(* IEC 61131-3 sources: TIA2AX/tests/test_projects/expected/HW_2200330_V18/ST40_PLC, 6 files *)

(* ---- HwInputs.st ---- *)
TYPE
	HwInputs : STRUCT
		ST40_2_DM260_Acquisition_Status_1 AT %B2500 : ARRAY[0..2] OF BYTE;
		ST40_2_DM260_Results_Status_1 AT %B2503 : BYTE;
		ST40_2_DM260_Soft_Event_Control_1 AT %B2504 : BYTE;
		ST40_2_DM260_Result_Data_64_bytes_1 AT %B2510 : ARRAY[0..71] OF BYTE;
		ST40_3_DM260_Acquisition_Status_1 AT %B3500 : ARRAY[0..2] OF BYTE;
		ST40_3_DM260_Results_Status_1 AT %B3503 : BYTE;
		ST40_3_DM260_Soft_Event_Control_1 AT %B3504 : BYTE;
		ST40_3_DM260_Result_Data_64_bytes_1 AT %B3510 : ARRAY[0..71] OF BYTE;
		ST40_1_DM260_Acquisition_Status_1 AT %B1600 : ARRAY[0..2] OF BYTE;
		ST40_1_DM260_Results_Status_1 AT %B1603 : BYTE;
		ST40_1_DM260_Soft_Event_Control_1 AT %B1604 : BYTE;
		ST40_1_DM260_Result_Data_64_bytes_1 AT %B1610 : ARRAY[0..71] OF BYTE;
		ST40_2_Promess_Menu_30_01_In_1 AT %B2100 : WORD;
		ST40_2_Promess_Menu_30_02_In_1 AT %B2102 : WORD;
		ST40_2_Promess_Menu_30_03_In_1 AT %B2104 : WORD;
		ST40_2_Promess_Menu_30_04_In_1 AT %B2106 : WORD;
		ST40_2_Promess_Menu_30_05_In_1 AT %B2108 : WORD;
		ST40_2_Promess_Menu_30_06_In_1 AT %B2110 : WORD;
		ST40_2_Promess_Menu_30_07_In_1 AT %B2112 : WORD;
		ST40_2_Promess_Menu_30_08_In_1 AT %B2114 : WORD;
		ST40_2_Promess_Menu_30_09_In_1 AT %B2116 : WORD;
		ST40_2_Promess_Menu_30_10_In_1 AT %B2118 : WORD;
		ST40_2_Promess_Menu_30_11_In_1 AT %B2120 : WORD;
		ST40_2_Promess_Menu_30_12_In_1 AT %B2122 : WORD;
		ST40_2_Promess_Menu_30_13_In_1 AT %B2124 : WORD;
		ST40_2_Promess_Menu_30_14_In_1 AT %B2126 : WORD;
		ST40_2_Promess_Menu_30_15_In_1 AT %B2128 : WORD;
		ST40_2_Promess_Menu_30_16_In_1 AT %B2130 : WORD;
		ST40_2_Promess_Menu_30_17_In_1 AT %B2132 : WORD;
		ST40_2_Promess_Menu_30_18_In_1 AT %B2134 : WORD;
		ST40_2_Promess_Menu_30_19_In_1 AT %B2136 : WORD;
		ST40_2_Promess_Menu_30_20_In_1 AT %B2138 : WORD;
		ST40_2_Promess_Menu_30_21_In_1 AT %B2140 : WORD;
		ST40_2_Promess_Menu_30_22_In_1 AT %B2142 : WORD;
		ST40_2_Promess_Menu_30_23_In_1 AT %B2144 : WORD;
		ST40_2_Promess_Menu_30_24_In_1 AT %B2146 : WORD;
		ST40_2_Promess_Menu_30_25_In_1 AT %B2148 : WORD;
		ST40_2_Promess_Menu_30_26_In_1 AT %B2150 : WORD;
		ST40_2_Promess_Menu_30_27_In_1 AT %B2152 : WORD;
		ST40_2_Promess_Menu_30_28_In_1 AT %B2154 : WORD;
		ST40_2_Promess_Menu_30_29_In_1 AT %B2156 : WORD;
		ST40_2_Promess_Menu_30_30_In_1 AT %B2158 : WORD;
		ST40_2_Promess_Menu_30_31_In_1 AT %B2160 : WORD;
		ST40_2_Promess_Menu_30_32_In_1 AT %B2162 : WORD;
		ST40_ET200SP_CM_4xIO_Link_1 AT %B100 : ARRAY[0..31] OF BYTE;
		ST40_ET200SP_CM_4xIO_Link_2 AT %B132 : ARRAY[0..31] OF BYTE;
		ST40_ET200SP_DI_8x24VDC_ST_1 AT %B0 : BYTE;
		ST40_ET200SP_DI_8x24VDC_ST_2 AT %B1 : BYTE;
		ST40_ET200SP_DI_16x24VDC_ST_1 AT %B2 : WORD;
		ST40_ET200SP_DI_8x24VDC_ST_3 AT %B4 : BYTE;
	END_STRUCT;
END_TYPE

(* ---- HwOutputs.st ---- *)
TYPE
	HwOutputs : STRUCT
		ST40_2_DM260_Acquisition_Control_1 AT %B2500 : BYTE;
		ST40_2_DM260_Results_Control_1 AT %B2503 : BYTE;
		ST40_2_DM260_Soft_Event_Control_1 AT %B2504 : BYTE;
		ST40_2_DM260_User_Data_64_bytes_1 AT %B2510 : ARRAY[0..67] OF BYTE;
		ST40_3_DM260_Acquisition_Control_1 AT %B3500 : BYTE;
		ST40_3_DM260_Results_Control_1 AT %B3503 : BYTE;
		ST40_3_DM260_Soft_Event_Control_1 AT %B3504 : BYTE;
		ST40_3_DM260_User_Data_64_bytes_1 AT %B3510 : ARRAY[0..67] OF BYTE;
		ST40_1_DM260_Acquisition_Control_1 AT %B1600 : BYTE;
		ST40_1_DM260_Results_Control_1 AT %B1603 : BYTE;
		ST40_1_DM260_Soft_Event_Control_1 AT %B1604 : BYTE;
		ST40_1_DM260_User_Data_64_bytes_1 AT %B1610 : ARRAY[0..67] OF BYTE;
		ST40_2_Promess_Menu_30_33_Out_1 AT %B2100 : WORD;
		ST40_2_Promess_Menu_30_34_Out_1 AT %B2102 : WORD;
		ST40_2_Promess_Menu_30_35_Out_1 AT %B2104 : WORD;
		ST40_2_Promess_Menu_30_36_Out_1 AT %B2106 : WORD;
		ST40_2_Promess_Menu_30_37_Out_1 AT %B2108 : WORD;
		ST40_2_Promess_Menu_30_38_Out_1 AT %B2110 : WORD;
		ST40_2_Promess_Menu_30_39_Out_1 AT %B2112 : WORD;
		ST40_2_Promess_Menu_30_40_Out_1 AT %B2114 : WORD;
		ST40_2_Promess_Menu_30_41_Out_1 AT %B2116 : WORD;
		ST40_2_Promess_Menu_30_42_Out_1 AT %B2118 : WORD;
		ST40_2_Promess_Menu_30_43_Out_1 AT %B2120 : WORD;
		ST40_2_Promess_Menu_30_44_Out_1 AT %B2122 : WORD;
		ST40_2_Promess_Menu_30_45_Out_1 AT %B2124 : WORD;
		ST40_2_Promess_Menu_30_46_Out_1 AT %B2126 : WORD;
		ST40_2_Promess_Menu_30_47_Out_1 AT %B2128 : WORD;
		ST40_2_Promess_Menu_30_48_Out_1 AT %B2130 : WORD;
		ST40_2_Promess_Menu_30_49_Out_1 AT %B2132 : WORD;
		ST40_2_Promess_Menu_30_50_Out_1 AT %B2134 : WORD;
		ST40_2_Promess_Menu_30_51_Out_1 AT %B2136 : WORD;
		ST40_2_Promess_Menu_30_52_Out_1 AT %B2138 : WORD;
		ST40_2_Promess_Menu_30_53_Out_1 AT %B2140 : WORD;
		ST40_2_Promess_Menu_30_54_Out_1 AT %B2142 : WORD;
		ST40_2_Promess_Menu_30_55_Out_1 AT %B2144 : WORD;
		ST40_2_Promess_Menu_30_56_Out_1 AT %B2146 : WORD;
		ST40_2_Promess_Menu_30_57_Out_1 AT %B2148 : WORD;
		ST40_2_Promess_Menu_30_58_Out_1 AT %B2150 : WORD;
		ST40_2_Promess_Menu_30_59_Out_1 AT %B2152 : WORD;
		ST40_2_Promess_Menu_30_60_Out_1 AT %B2154 : WORD;
		ST40_2_Promess_Menu_30_61_Out_1 AT %B2156 : WORD;
		ST40_2_Promess_Menu_30_62_Out_1 AT %B2158 : WORD;
		ST40_2_Promess_Menu_30_63_Out_1 AT %B2160 : WORD;
		ST40_2_Promess_Menu_30_64_Out_1 AT %B2162 : WORD;
		ST40_CPX_MPA1S_VMPA1_FB_EMS_8_8DO_1 AT %B200 : BYTE;
		ST40_CPX_MPA1S_VMPA1_FB_EMS_8_8DO_2 AT %B201 : BYTE;
		ST40_CPX_MPA1S_VMPA1_FB_EMS_8_8DO_3 AT %B202 : BYTE;
		ST40_CPX_MPA1G_VMPA1_FB_EMG_8_8DO_1 AT %B203 : BYTE;
		ST40_ET200SP_CM_4xIO_Link_1 AT %B100 : ARRAY[0..31] OF BYTE;
		ST40_ET200SP_CM_4xIO_Link_2 AT %B132 : ARRAY[0..31] OF BYTE;
		ST40_ET200SP_DQ_16x24VDC_0_5A_ST_1 AT %B0 : WORD;
		ST40_ET200SP_DQ_8x24VDC_0_5A_ST_2 AT %B2 : BYTE;
		ST40_ET200SP_DQ_8x24VDC_0_5A_ST_3 AT %B3 : BYTE;
	END_STRUCT;
END_TYPE

(* ---- PlcInputs.st ---- *)
TYPE
	PlcInputs : STRUCT
		ST40_2_DM260_Acquisition_Status_1 : ARRAY[0..2] OF BYTE;
		ST40_2_DM260_Results_Status_1 : BYTE;
		ST40_2_DM260_Soft_Event_Control_1 : BYTE;
		ST40_2_DM260_Result_Data_64_bytes_1 : ARRAY[0..71] OF BYTE;
		ST40_3_DM260_Acquisition_Status_1 : ARRAY[0..2] OF BYTE;
		ST40_3_DM260_Results_Status_1 : BYTE;
		ST40_3_DM260_Soft_Event_Control_1 : BYTE;
		ST40_3_DM260_Result_Data_64_bytes_1 : ARRAY[0..71] OF BYTE;
		ST40_1_DM260_Acquisition_Status_1 : ARRAY[0..2] OF BYTE;
		ST40_1_DM260_Results_Status_1 : BYTE;
		ST40_1_DM260_Soft_Event_Control_1 : BYTE;
		ST40_1_DM260_Result_Data_64_bytes_1 : ARRAY[0..71] OF BYTE;
		ST40_2_Promess_Menu_30_01_In_1 : WORD;
		ST40_2_Promess_Menu_30_02_In_1 : WORD;
		ST40_2_Promess_Menu_30_03_In_1 : WORD;
		ST40_2_Promess_Menu_30_04_In_1 : WORD;
		ST40_2_Promess_Menu_30_05_In_1 : WORD;
		ST40_2_Promess_Menu_30_06_In_1 : WORD;
		ST40_2_Promess_Menu_30_07_In_1 : WORD;
		ST40_2_Promess_Menu_30_08_In_1 : WORD;
		ST40_2_Promess_Menu_30_09_In_1 : WORD;
		ST40_2_Promess_Menu_30_10_In_1 : WORD;
		ST40_2_Promess_Menu_30_11_In_1 : WORD;
		ST40_2_Promess_Menu_30_12_In_1 : WORD;
		ST40_2_Promess_Menu_30_13_In_1 : WORD;
		ST40_2_Promess_Menu_30_14_In_1 : WORD;
		ST40_2_Promess_Menu_30_15_In_1 : WORD;
		ST40_2_Promess_Menu_30_16_In_1 : WORD;
		ST40_2_Promess_Menu_30_17_In_1 : WORD;
		ST40_2_Promess_Menu_30_18_In_1 : WORD;
		ST40_2_Promess_Menu_30_19_In_1 : WORD;
		ST40_2_Promess_Menu_30_20_In_1 : WORD;
		ST40_2_Promess_Menu_30_21_In_1 : WORD;
		ST40_2_Promess_Menu_30_22_In_1 : WORD;
		ST40_2_Promess_Menu_30_23_In_1 : WORD;
		ST40_2_Promess_Menu_30_24_In_1 : WORD;
		ST40_2_Promess_Menu_30_25_In_1 : WORD;
		ST40_2_Promess_Menu_30_26_In_1 : WORD;
		ST40_2_Promess_Menu_30_27_In_1 : WORD;
		ST40_2_Promess_Menu_30_28_In_1 : WORD;
		ST40_2_Promess_Menu_30_29_In_1 : WORD;
		ST40_2_Promess_Menu_30_30_In_1 : WORD;
		ST40_2_Promess_Menu_30_31_In_1 : WORD;
		ST40_2_Promess_Menu_30_32_In_1 : WORD;
		ST40_ET200SP_CM_4xIO_Link_1 : ARRAY[0..31] OF BYTE;
		ST40_ET200SP_CM_4xIO_Link_2 : ARRAY[0..31] OF BYTE;
		ST40_ET200SP_DI_8x24VDC_ST_1 : BYTE;
		ST40_ET200SP_DI_8x24VDC_ST_2 : BYTE;
		ST40_ET200SP_DI_16x24VDC_ST_1 : WORD;
		ST40_ET200SP_DI_8x24VDC_ST_3 : BYTE;
	END_STRUCT;
END_TYPE

(* ---- PlcOutputs.st ---- *)
TYPE
	PlcOutputs : STRUCT
		ST40_2_DM260_Acquisition_Control_1 : BYTE;
		ST40_2_DM260_Results_Control_1 : BYTE;
		ST40_2_DM260_Soft_Event_Control_1 : BYTE;
		ST40_2_DM260_User_Data_64_bytes_1 : ARRAY[0..67] OF BYTE;
		ST40_3_DM260_Acquisition_Control_1 : BYTE;
		ST40_3_DM260_Results_Control_1 : BYTE;
		ST40_3_DM260_Soft_Event_Control_1 : BYTE;
		ST40_3_DM260_User_Data_64_bytes_1 : ARRAY[0..67] OF BYTE;
		ST40_1_DM260_Acquisition_Control_1 : BYTE;
		ST40_1_DM260_Results_Control_1 : BYTE;
		ST40_1_DM260_Soft_Event_Control_1 : BYTE;
		ST40_1_DM260_User_Data_64_bytes_1 : ARRAY[0..67] OF BYTE;
		ST40_2_Promess_Menu_30_33_Out_1 : WORD;
		ST40_2_Promess_Menu_30_34_Out_1 : WORD;
		ST40_2_Promess_Menu_30_35_Out_1 : WORD;
		ST40_2_Promess_Menu_30_36_Out_1 : WORD;
		ST40_2_Promess_Menu_30_37_Out_1 : WORD;
		ST40_2_Promess_Menu_30_38_Out_1 : WORD;
		ST40_2_Promess_Menu_30_39_Out_1 : WORD;
		ST40_2_Promess_Menu_30_40_Out_1 : WORD;
		ST40_2_Promess_Menu_30_41_Out_1 : WORD;
		ST40_2_Promess_Menu_30_42_Out_1 : WORD;
		ST40_2_Promess_Menu_30_43_Out_1 : WORD;
		ST40_2_Promess_Menu_30_44_Out_1 : WORD;
		ST40_2_Promess_Menu_30_45_Out_1 : WORD;
		ST40_2_Promess_Menu_30_46_Out_1 : WORD;
		ST40_2_Promess_Menu_30_47_Out_1 : WORD;
		ST40_2_Promess_Menu_30_48_Out_1 : WORD;
		ST40_2_Promess_Menu_30_49_Out_1 : WORD;
		ST40_2_Promess_Menu_30_50_Out_1 : WORD;
		ST40_2_Promess_Menu_30_51_Out_1 : WORD;
		ST40_2_Promess_Menu_30_52_Out_1 : WORD;
		ST40_2_Promess_Menu_30_53_Out_1 : WORD;
		ST40_2_Promess_Menu_30_54_Out_1 : WORD;
		ST40_2_Promess_Menu_30_55_Out_1 : WORD;
		ST40_2_Promess_Menu_30_56_Out_1 : WORD;
		ST40_2_Promess_Menu_30_57_Out_1 : WORD;
		ST40_2_Promess_Menu_30_58_Out_1 : WORD;
		ST40_2_Promess_Menu_30_59_Out_1 : WORD;
		ST40_2_Promess_Menu_30_60_Out_1 : WORD;
		ST40_2_Promess_Menu_30_61_Out_1 : WORD;
		ST40_2_Promess_Menu_30_62_Out_1 : WORD;
		ST40_2_Promess_Menu_30_63_Out_1 : WORD;
		ST40_2_Promess_Menu_30_64_Out_1 : WORD;
		ST40_CPX_MPA1S_VMPA1_FB_EMS_8_8DO_1 : BYTE;
		ST40_CPX_MPA1S_VMPA1_FB_EMS_8_8DO_2 : BYTE;
		ST40_CPX_MPA1S_VMPA1_FB_EMS_8_8DO_3 : BYTE;
		ST40_CPX_MPA1G_VMPA1_FB_EMG_8_8DO_1 : BYTE;
		ST40_ET200SP_CM_4xIO_Link_1 : ARRAY[0..31] OF BYTE;
		ST40_ET200SP_CM_4xIO_Link_2 : ARRAY[0..31] OF BYTE;
		ST40_ET200SP_DQ_16x24VDC_0_5A_ST_1 : WORD;
		ST40_ET200SP_DQ_8x24VDC_0_5A_ST_2 : BYTE;
		ST40_ET200SP_DQ_8x24VDC_0_5A_ST_3 : BYTE;
	END_STRUCT;
END_TYPE

(* ---- CopyInputs.st ---- *)
FUNCTION CopyInputs
	VAR_EXTERNAL
		HwInputs : HwInputs;
		PlcInputs : PlcInputs;
	END_VAR
	PlcInputs.ST40_2_DM260_Acquisition_Status_1[0] := HwInputs.ST40_2_DM260_Acquisition_Status_1[0];
	PlcInputs.ST40_2_DM260_Acquisition_Status_1[1] := HwInputs.ST40_2_DM260_Acquisition_Status_1[1];
	PlcInputs.ST40_2_DM260_Acquisition_Status_1[2] := HwInputs.ST40_2_DM260_Acquisition_Status_1[2];
	PlcInputs.ST40_2_DM260_Results_Status_1 := HwInputs.ST40_2_DM260_Results_Status_1;
	PlcInputs.ST40_2_DM260_Soft_Event_Control_1 := HwInputs.ST40_2_DM260_Soft_Event_Control_1;
	PlcInputs.ST40_2_DM260_Result_Data_64_bytes_1[0] := HwInputs.ST40_2_DM260_Result_Data_64_bytes_1[0];
	PlcInputs.ST40_2_DM260_Result_Data_64_bytes_1[1] := HwInputs.ST40_2_DM260_Result_Data_64_bytes_1[1];
	PlcInputs.ST40_2_DM260_Result_Data_64_bytes_1[2] := HwInputs.ST40_2_DM260_Result_Data_64_bytes_1[2];
	PlcInputs.ST40_2_DM260_Result_Data_64_bytes_1[3] := HwInputs.ST40_2_DM260_Result_Data_64_bytes_1[3];
	PlcInputs.ST40_2_DM260_Result_Data_64_bytes_1[4] := HwInputs.ST40_2_DM260_Result_Data_64_bytes_1[4];
	PlcInputs.ST40_2_DM260_Result_Data_64_bytes_1[5] := HwInputs.ST40_2_DM260_Result_Data_64_bytes_1[5];
	PlcInputs.ST40_2_DM260_Result_Data_64_bytes_1[6] := HwInputs.ST40_2_DM260_Result_Data_64_bytes_1[6];
	PlcInputs.ST40_2_DM260_Result_Data_64_bytes_1[7] := HwInputs.ST40_2_DM260_Result_Data_64_bytes_1[7];
	PlcInputs.ST40_2_DM260_Result_Data_64_bytes_1[8] := HwInputs.ST40_2_DM260_Result_Data_64_bytes_1[8];
	PlcInputs.ST40_2_DM260_Result_Data_64_bytes_1[9] := HwInputs.ST40_2_DM260_Result_Data_64_bytes_1[9];
	PlcInputs.ST40_2_DM260_Result_Data_64_bytes_1[10] := HwInputs.ST40_2_DM260_Result_Data_64_bytes_1[10];
	PlcInputs.ST40_2_DM260_Result_Data_64_bytes_1[11] := HwInputs.ST40_2_DM260_Result_Data_64_bytes_1[11];
	PlcInputs.ST40_2_DM260_Result_Data_64_bytes_1[12] := HwInputs.ST40_2_DM260_Result_Data_64_bytes_1[12];
	PlcInputs.ST40_2_DM260_Result_Data_64_bytes_1[13] := HwInputs.ST40_2_DM260_Result_Data_64_bytes_1[13];
	PlcInputs.ST40_2_DM260_Result_Data_64_bytes_1[14] := HwInputs.ST40_2_DM260_Result_Data_64_bytes_1[14];
	PlcInputs.ST40_2_DM260_Result_Data_64_bytes_1[15] := HwInputs.ST40_2_DM260_Result_Data_64_bytes_1[15];
	PlcInputs.ST40_2_DM260_Result_Data_64_bytes_1[16] := HwInputs.ST40_2_DM260_Result_Data_64_bytes_1[16];
	PlcInputs.ST40_2_DM260_Result_Data_64_bytes_1[17] := HwInputs.ST40_2_DM260_Result_Data_64_bytes_1[17];
	PlcInputs.ST40_2_DM260_Result_Data_64_bytes_1[18] := HwInputs.ST40_2_DM260_Result_Data_64_bytes_1[18];
	PlcInputs.ST40_2_DM260_Result_Data_64_bytes_1[19] := HwInputs.ST40_2_DM260_Result_Data_64_bytes_1[19];
	PlcInputs.ST40_2_DM260_Result_Data_64_bytes_1[20] := HwInputs.ST40_2_DM260_Result_Data_64_bytes_1[20];
	PlcInputs.ST40_2_DM260_Result_Data_64_bytes_1[21] := HwInputs.ST40_2_DM260_Result_Data_64_bytes_1[21];
	PlcInputs.ST40_2_DM260_Result_Data_64_bytes_1[22] := HwInputs.ST40_2_DM260_Result_Data_64_bytes_1[22];
	PlcInputs.ST40_2_DM260_Result_Data_64_bytes_1[23] := HwInputs.ST40_2_DM260_Result_Data_64_bytes_1[23];
	PlcInputs.ST40_2_DM260_Result_Data_64_bytes_1[24] := HwInputs.ST40_2_DM260_Result_Data_64_bytes_1[24];
	PlcInputs.ST40_2_DM260_Result_Data_64_bytes_1[25] := HwInputs.ST40_2_DM260_Result_Data_64_bytes_1[25];
	PlcInputs.ST40_2_DM260_Result_Data_64_bytes_1[26] := HwInputs.ST40_2_DM260_Result_Data_64_bytes_1[26];
	PlcInputs.ST40_2_DM260_Result_Data_64_bytes_1[27] := HwInputs.ST40_2_DM260_Result_Data_64_bytes_1[27];
	PlcInputs.ST40_2_DM260_Result_Data_64_bytes_1[28] := HwInputs.ST40_2_DM260_Result_Data_64_bytes_1[28];
	PlcInputs.ST40_2_DM260_Result_Data_64_bytes_1[29] := HwInputs.ST40_2_DM260_Result_Data_64_bytes_1[29];
	PlcInputs.ST40_2_DM260_Result_Data_64_bytes_1[30] := HwInputs.ST40_2_DM260_Result_Data_64_bytes_1[30];
	PlcInputs.ST40_2_DM260_Result_Data_64_bytes_1[31] := HwInputs.ST40_2_DM260_Result_Data_64_bytes_1[31];
	PlcInputs.ST40_2_DM260_Result_Data_64_bytes_1[32] := HwInputs.ST40_2_DM260_Result_Data_64_bytes_1[32];
	PlcInputs.ST40_2_DM260_Result_Data_64_bytes_1[33] := HwInputs.ST40_2_DM260_Result_Data_64_bytes_1[33];
	PlcInputs.ST40_2_DM260_Result_Data_64_bytes_1[34] := HwInputs.ST40_2_DM260_Result_Data_64_bytes_1[34];
	PlcInputs.ST40_2_DM260_Result_Data_64_bytes_1[35] := HwInputs.ST40_2_DM260_Result_Data_64_bytes_1[35];
	PlcInputs.ST40_2_DM260_Result_Data_64_bytes_1[36] := HwInputs.ST40_2_DM260_Result_Data_64_bytes_1[36];
	PlcInputs.ST40_2_DM260_Result_Data_64_bytes_1[37] := HwInputs.ST40_2_DM260_Result_Data_64_bytes_1[37];
	PlcInputs.ST40_2_DM260_Result_Data_64_bytes_1[38] := HwInputs.ST40_2_DM260_Result_Data_64_bytes_1[38];
	PlcInputs.ST40_2_DM260_Result_Data_64_bytes_1[39] := HwInputs.ST40_2_DM260_Result_Data_64_bytes_1[39];
	PlcInputs.ST40_2_DM260_Result_Data_64_bytes_1[40] := HwInputs.ST40_2_DM260_Result_Data_64_bytes_1[40];
	PlcInputs.ST40_2_DM260_Result_Data_64_bytes_1[41] := HwInputs.ST40_2_DM260_Result_Data_64_bytes_1[41];
	PlcInputs.ST40_2_DM260_Result_Data_64_bytes_1[42] := HwInputs.ST40_2_DM260_Result_Data_64_bytes_1[42];
	PlcInputs.ST40_2_DM260_Result_Data_64_bytes_1[43] := HwInputs.ST40_2_DM260_Result_Data_64_bytes_1[43];
	PlcInputs.ST40_2_DM260_Result_Data_64_bytes_1[44] := HwInputs.ST40_2_DM260_Result_Data_64_bytes_1[44];
	PlcInputs.ST40_2_DM260_Result_Data_64_bytes_1[45] := HwInputs.ST40_2_DM260_Result_Data_64_bytes_1[45];
	PlcInputs.ST40_2_DM260_Result_Data_64_bytes_1[46] := HwInputs.ST40_2_DM260_Result_Data_64_bytes_1[46];
	PlcInputs.ST40_2_DM260_Result_Data_64_bytes_1[47] := HwInputs.ST40_2_DM260_Result_Data_64_bytes_1[47];
	PlcInputs.ST40_2_DM260_Result_Data_64_bytes_1[48] := HwInputs.ST40_2_DM260_Result_Data_64_bytes_1[48];
	PlcInputs.ST40_2_DM260_Result_Data_64_bytes_1[49] := HwInputs.ST40_2_DM260_Result_Data_64_bytes_1[49];
	PlcInputs.ST40_2_DM260_Result_Data_64_bytes_1[50] := HwInputs.ST40_2_DM260_Result_Data_64_bytes_1[50];
	PlcInputs.ST40_2_DM260_Result_Data_64_bytes_1[51] := HwInputs.ST40_2_DM260_Result_Data_64_bytes_1[51];
	PlcInputs.ST40_2_DM260_Result_Data_64_bytes_1[52] := HwInputs.ST40_2_DM260_Result_Data_64_bytes_1[52];
	PlcInputs.ST40_2_DM260_Result_Data_64_bytes_1[53] := HwInputs.ST40_2_DM260_Result_Data_64_bytes_1[53];
	PlcInputs.ST40_2_DM260_Result_Data_64_bytes_1[54] := HwInputs.ST40_2_DM260_Result_Data_64_bytes_1[54];
	PlcInputs.ST40_2_DM260_Result_Data_64_bytes_1[55] := HwInputs.ST40_2_DM260_Result_Data_64_bytes_1[55];
	PlcInputs.ST40_2_DM260_Result_Data_64_bytes_1[56] := HwInputs.ST40_2_DM260_Result_Data_64_bytes_1[56];
	PlcInputs.ST40_2_DM260_Result_Data_64_bytes_1[57] := HwInputs.ST40_2_DM260_Result_Data_64_bytes_1[57];
	PlcInputs.ST40_2_DM260_Result_Data_64_bytes_1[58] := HwInputs.ST40_2_DM260_Result_Data_64_bytes_1[58];
	PlcInputs.ST40_2_DM260_Result_Data_64_bytes_1[59] := HwInputs.ST40_2_DM260_Result_Data_64_bytes_1[59];
	PlcInputs.ST40_2_DM260_Result_Data_64_bytes_1[60] := HwInputs.ST40_2_DM260_Result_Data_64_bytes_1[60];
	PlcInputs.ST40_2_DM260_Result_Data_64_bytes_1[61] := HwInputs.ST40_2_DM260_Result_Data_64_bytes_1[61];
	PlcInputs.ST40_2_DM260_Result_Data_64_bytes_1[62] := HwInputs.ST40_2_DM260_Result_Data_64_bytes_1[62];
	PlcInputs.ST40_2_DM260_Result_Data_64_bytes_1[63] := HwInputs.ST40_2_DM260_Result_Data_64_bytes_1[63];
	PlcInputs.ST40_2_DM260_Result_Data_64_bytes_1[64] := HwInputs.ST40_2_DM260_Result_Data_64_bytes_1[64];
	PlcInputs.ST40_2_DM260_Result_Data_64_bytes_1[65] := HwInputs.ST40_2_DM260_Result_Data_64_bytes_1[65];
	PlcInputs.ST40_2_DM260_Result_Data_64_bytes_1[66] := HwInputs.ST40_2_DM260_Result_Data_64_bytes_1[66];
	PlcInputs.ST40_2_DM260_Result_Data_64_bytes_1[67] := HwInputs.ST40_2_DM260_Result_Data_64_bytes_1[67];
	PlcInputs.ST40_2_DM260_Result_Data_64_bytes_1[68] := HwInputs.ST40_2_DM260_Result_Data_64_bytes_1[68];
	PlcInputs.ST40_2_DM260_Result_Data_64_bytes_1[69] := HwInputs.ST40_2_DM260_Result_Data_64_bytes_1[69];
	PlcInputs.ST40_2_DM260_Result_Data_64_bytes_1[70] := HwInputs.ST40_2_DM260_Result_Data_64_bytes_1[70];
	PlcInputs.ST40_2_DM260_Result_Data_64_bytes_1[71] := HwInputs.ST40_2_DM260_Result_Data_64_bytes_1[71];
	PlcInputs.ST40_3_DM260_Acquisition_Status_1[0] := HwInputs.ST40_3_DM260_Acquisition_Status_1[0];
	PlcInputs.ST40_3_DM260_Acquisition_Status_1[1] := HwInputs.ST40_3_DM260_Acquisition_Status_1[1];
	PlcInputs.ST40_3_DM260_Acquisition_Status_1[2] := HwInputs.ST40_3_DM260_Acquisition_Status_1[2];
	PlcInputs.ST40_3_DM260_Results_Status_1 := HwInputs.ST40_3_DM260_Results_Status_1;
	PlcInputs.ST40_3_DM260_Soft_Event_Control_1 := HwInputs.ST40_3_DM260_Soft_Event_Control_1;
	PlcInputs.ST40_3_DM260_Result_Data_64_bytes_1[0] := HwInputs.ST40_3_DM260_Result_Data_64_bytes_1[0];
	PlcInputs.ST40_3_DM260_Result_Data_64_bytes_1[1] := HwInputs.ST40_3_DM260_Result_Data_64_bytes_1[1];
	PlcInputs.ST40_3_DM260_Result_Data_64_bytes_1[2] := HwInputs.ST40_3_DM260_Result_Data_64_bytes_1[2];
	PlcInputs.ST40_3_DM260_Result_Data_64_bytes_1[3] := HwInputs.ST40_3_DM260_Result_Data_64_bytes_1[3];
	PlcInputs.ST40_3_DM260_Result_Data_64_bytes_1[4] := HwInputs.ST40_3_DM260_Result_Data_64_bytes_1[4];
	PlcInputs.ST40_3_DM260_Result_Data_64_bytes_1[5] := HwInputs.ST40_3_DM260_Result_Data_64_bytes_1[5];
	PlcInputs.ST40_3_DM260_Result_Data_64_bytes_1[6] := HwInputs.ST40_3_DM260_Result_Data_64_bytes_1[6];
	PlcInputs.ST40_3_DM260_Result_Data_64_bytes_1[7] := HwInputs.ST40_3_DM260_Result_Data_64_bytes_1[7];
	PlcInputs.ST40_3_DM260_Result_Data_64_bytes_1[8] := HwInputs.ST40_3_DM260_Result_Data_64_bytes_1[8];
	PlcInputs.ST40_3_DM260_Result_Data_64_bytes_1[9] := HwInputs.ST40_3_DM260_Result_Data_64_bytes_1[9];
	PlcInputs.ST40_3_DM260_Result_Data_64_bytes_1[10] := HwInputs.ST40_3_DM260_Result_Data_64_bytes_1[10];
	PlcInputs.ST40_3_DM260_Result_Data_64_bytes_1[11] := HwInputs.ST40_3_DM260_Result_Data_64_bytes_1[11];
	PlcInputs.ST40_3_DM260_Result_Data_64_bytes_1[12] := HwInputs.ST40_3_DM260_Result_Data_64_bytes_1[12];
	PlcInputs.ST40_3_DM260_Result_Data_64_bytes_1[13] := HwInputs.ST40_3_DM260_Result_Data_64_bytes_1[13];
	PlcInputs.ST40_3_DM260_Result_Data_64_bytes_1[14] := HwInputs.ST40_3_DM260_Result_Data_64_bytes_1[14];
	PlcInputs.ST40_3_DM260_Result_Data_64_bytes_1[15] := HwInputs.ST40_3_DM260_Result_Data_64_bytes_1[15];
	PlcInputs.ST40_3_DM260_Result_Data_64_bytes_1[16] := HwInputs.ST40_3_DM260_Result_Data_64_bytes_1[16];
	PlcInputs.ST40_3_DM260_Result_Data_64_bytes_1[17] := HwInputs.ST40_3_DM260_Result_Data_64_bytes_1[17];
	PlcInputs.ST40_3_DM260_Result_Data_64_bytes_1[18] := HwInputs.ST40_3_DM260_Result_Data_64_bytes_1[18];
	PlcInputs.ST40_3_DM260_Result_Data_64_bytes_1[19] := HwInputs.ST40_3_DM260_Result_Data_64_bytes_1[19];
	PlcInputs.ST40_3_DM260_Result_Data_64_bytes_1[20] := HwInputs.ST40_3_DM260_Result_Data_64_bytes_1[20];
	PlcInputs.ST40_3_DM260_Result_Data_64_bytes_1[21] := HwInputs.ST40_3_DM260_Result_Data_64_bytes_1[21];
	PlcInputs.ST40_3_DM260_Result_Data_64_bytes_1[22] := HwInputs.ST40_3_DM260_Result_Data_64_bytes_1[22];
	PlcInputs.ST40_3_DM260_Result_Data_64_bytes_1[23] := HwInputs.ST40_3_DM260_Result_Data_64_bytes_1[23];
	PlcInputs.ST40_3_DM260_Result_Data_64_bytes_1[24] := HwInputs.ST40_3_DM260_Result_Data_64_bytes_1[24];
	PlcInputs.ST40_3_DM260_Result_Data_64_bytes_1[25] := HwInputs.ST40_3_DM260_Result_Data_64_bytes_1[25];
	PlcInputs.ST40_3_DM260_Result_Data_64_bytes_1[26] := HwInputs.ST40_3_DM260_Result_Data_64_bytes_1[26];
	PlcInputs.ST40_3_DM260_Result_Data_64_bytes_1[27] := HwInputs.ST40_3_DM260_Result_Data_64_bytes_1[27];
	PlcInputs.ST40_3_DM260_Result_Data_64_bytes_1[28] := HwInputs.ST40_3_DM260_Result_Data_64_bytes_1[28];
	PlcInputs.ST40_3_DM260_Result_Data_64_bytes_1[29] := HwInputs.ST40_3_DM260_Result_Data_64_bytes_1[29];
	PlcInputs.ST40_3_DM260_Result_Data_64_bytes_1[30] := HwInputs.ST40_3_DM260_Result_Data_64_bytes_1[30];
	PlcInputs.ST40_3_DM260_Result_Data_64_bytes_1[31] := HwInputs.ST40_3_DM260_Result_Data_64_bytes_1[31];
	PlcInputs.ST40_3_DM260_Result_Data_64_bytes_1[32] := HwInputs.ST40_3_DM260_Result_Data_64_bytes_1[32];
	PlcInputs.ST40_3_DM260_Result_Data_64_bytes_1[33] := HwInputs.ST40_3_DM260_Result_Data_64_bytes_1[33];
	PlcInputs.ST40_3_DM260_Result_Data_64_bytes_1[34] := HwInputs.ST40_3_DM260_Result_Data_64_bytes_1[34];
	PlcInputs.ST40_3_DM260_Result_Data_64_bytes_1[35] := HwInputs.ST40_3_DM260_Result_Data_64_bytes_1[35];
	PlcInputs.ST40_3_DM260_Result_Data_64_bytes_1[36] := HwInputs.ST40_3_DM260_Result_Data_64_bytes_1[36];
	PlcInputs.ST40_3_DM260_Result_Data_64_bytes_1[37] := HwInputs.ST40_3_DM260_Result_Data_64_bytes_1[37];
	PlcInputs.ST40_3_DM260_Result_Data_64_bytes_1[38] := HwInputs.ST40_3_DM260_Result_Data_64_bytes_1[38];
	PlcInputs.ST40_3_DM260_Result_Data_64_bytes_1[39] := HwInputs.ST40_3_DM260_Result_Data_64_bytes_1[39];
	PlcInputs.ST40_3_DM260_Result_Data_64_bytes_1[40] := HwInputs.ST40_3_DM260_Result_Data_64_bytes_1[40];
	PlcInputs.ST40_3_DM260_Result_Data_64_bytes_1[41] := HwInputs.ST40_3_DM260_Result_Data_64_bytes_1[41];
	PlcInputs.ST40_3_DM260_Result_Data_64_bytes_1[42] := HwInputs.ST40_3_DM260_Result_Data_64_bytes_1[42];
	PlcInputs.ST40_3_DM260_Result_Data_64_bytes_1[43] := HwInputs.ST40_3_DM260_Result_Data_64_bytes_1[43];
	PlcInputs.ST40_3_DM260_Result_Data_64_bytes_1[44] := HwInputs.ST40_3_DM260_Result_Data_64_bytes_1[44];
	PlcInputs.ST40_3_DM260_Result_Data_64_bytes_1[45] := HwInputs.ST40_3_DM260_Result_Data_64_bytes_1[45];
	PlcInputs.ST40_3_DM260_Result_Data_64_bytes_1[46] := HwInputs.ST40_3_DM260_Result_Data_64_bytes_1[46];
	PlcInputs.ST40_3_DM260_Result_Data_64_bytes_1[47] := HwInputs.ST40_3_DM260_Result_Data_64_bytes_1[47];
	PlcInputs.ST40_3_DM260_Result_Data_64_bytes_1[48] := HwInputs.ST40_3_DM260_Result_Data_64_bytes_1[48];
	PlcInputs.ST40_3_DM260_Result_Data_64_bytes_1[49] := HwInputs.ST40_3_DM260_Result_Data_64_bytes_1[49];
	PlcInputs.ST40_3_DM260_Result_Data_64_bytes_1[50] := HwInputs.ST40_3_DM260_Result_Data_64_bytes_1[50];
	PlcInputs.ST40_3_DM260_Result_Data_64_bytes_1[51] := HwInputs.ST40_3_DM260_Result_Data_64_bytes_1[51];
	PlcInputs.ST40_3_DM260_Result_Data_64_bytes_1[52] := HwInputs.ST40_3_DM260_Result_Data_64_bytes_1[52];
	PlcInputs.ST40_3_DM260_Result_Data_64_bytes_1[53] := HwInputs.ST40_3_DM260_Result_Data_64_bytes_1[53];
	PlcInputs.ST40_3_DM260_Result_Data_64_bytes_1[54] := HwInputs.ST40_3_DM260_Result_Data_64_bytes_1[54];
	PlcInputs.ST40_3_DM260_Result_Data_64_bytes_1[55] := HwInputs.ST40_3_DM260_Result_Data_64_bytes_1[55];
	PlcInputs.ST40_3_DM260_Result_Data_64_bytes_1[56] := HwInputs.ST40_3_DM260_Result_Data_64_bytes_1[56];
	PlcInputs.ST40_3_DM260_Result_Data_64_bytes_1[57] := HwInputs.ST40_3_DM260_Result_Data_64_bytes_1[57];
	PlcInputs.ST40_3_DM260_Result_Data_64_bytes_1[58] := HwInputs.ST40_3_DM260_Result_Data_64_bytes_1[58];
	PlcInputs.ST40_3_DM260_Result_Data_64_bytes_1[59] := HwInputs.ST40_3_DM260_Result_Data_64_bytes_1[59];
	PlcInputs.ST40_3_DM260_Result_Data_64_bytes_1[60] := HwInputs.ST40_3_DM260_Result_Data_64_bytes_1[60];
	PlcInputs.ST40_3_DM260_Result_Data_64_bytes_1[61] := HwInputs.ST40_3_DM260_Result_Data_64_bytes_1[61];
	PlcInputs.ST40_3_DM260_Result_Data_64_bytes_1[62] := HwInputs.ST40_3_DM260_Result_Data_64_bytes_1[62];
	PlcInputs.ST40_3_DM260_Result_Data_64_bytes_1[63] := HwInputs.ST40_3_DM260_Result_Data_64_bytes_1[63];
	PlcInputs.ST40_3_DM260_Result_Data_64_bytes_1[64] := HwInputs.ST40_3_DM260_Result_Data_64_bytes_1[64];
	PlcInputs.ST40_3_DM260_Result_Data_64_bytes_1[65] := HwInputs.ST40_3_DM260_Result_Data_64_bytes_1[65];
	PlcInputs.ST40_3_DM260_Result_Data_64_bytes_1[66] := HwInputs.ST40_3_DM260_Result_Data_64_bytes_1[66];
	PlcInputs.ST40_3_DM260_Result_Data_64_bytes_1[67] := HwInputs.ST40_3_DM260_Result_Data_64_bytes_1[67];
	PlcInputs.ST40_3_DM260_Result_Data_64_bytes_1[68] := HwInputs.ST40_3_DM260_Result_Data_64_bytes_1[68];
	PlcInputs.ST40_3_DM260_Result_Data_64_bytes_1[69] := HwInputs.ST40_3_DM260_Result_Data_64_bytes_1[69];
	PlcInputs.ST40_3_DM260_Result_Data_64_bytes_1[70] := HwInputs.ST40_3_DM260_Result_Data_64_bytes_1[70];
	PlcInputs.ST40_3_DM260_Result_Data_64_bytes_1[71] := HwInputs.ST40_3_DM260_Result_Data_64_bytes_1[71];
	PlcInputs.ST40_1_DM260_Acquisition_Status_1[0] := HwInputs.ST40_1_DM260_Acquisition_Status_1[0];
	PlcInputs.ST40_1_DM260_Acquisition_Status_1[1] := HwInputs.ST40_1_DM260_Acquisition_Status_1[1];
	PlcInputs.ST40_1_DM260_Acquisition_Status_1[2] := HwInputs.ST40_1_DM260_Acquisition_Status_1[2];
	PlcInputs.ST40_1_DM260_Results_Status_1 := HwInputs.ST40_1_DM260_Results_Status_1;
	PlcInputs.ST40_1_DM260_Soft_Event_Control_1 := HwInputs.ST40_1_DM260_Soft_Event_Control_1;
	PlcInputs.ST40_1_DM260_Result_Data_64_bytes_1[0] := HwInputs.ST40_1_DM260_Result_Data_64_bytes_1[0];
	PlcInputs.ST40_1_DM260_Result_Data_64_bytes_1[1] := HwInputs.ST40_1_DM260_Result_Data_64_bytes_1[1];
	PlcInputs.ST40_1_DM260_Result_Data_64_bytes_1[2] := HwInputs.ST40_1_DM260_Result_Data_64_bytes_1[2];
	PlcInputs.ST40_1_DM260_Result_Data_64_bytes_1[3] := HwInputs.ST40_1_DM260_Result_Data_64_bytes_1[3];
	PlcInputs.ST40_1_DM260_Result_Data_64_bytes_1[4] := HwInputs.ST40_1_DM260_Result_Data_64_bytes_1[4];
	PlcInputs.ST40_1_DM260_Result_Data_64_bytes_1[5] := HwInputs.ST40_1_DM260_Result_Data_64_bytes_1[5];
	PlcInputs.ST40_1_DM260_Result_Data_64_bytes_1[6] := HwInputs.ST40_1_DM260_Result_Data_64_bytes_1[6];
	PlcInputs.ST40_1_DM260_Result_Data_64_bytes_1[7] := HwInputs.ST40_1_DM260_Result_Data_64_bytes_1[7];
	PlcInputs.ST40_1_DM260_Result_Data_64_bytes_1[8] := HwInputs.ST40_1_DM260_Result_Data_64_bytes_1[8];
	PlcInputs.ST40_1_DM260_Result_Data_64_bytes_1[9] := HwInputs.ST40_1_DM260_Result_Data_64_bytes_1[9];
	PlcInputs.ST40_1_DM260_Result_Data_64_bytes_1[10] := HwInputs.ST40_1_DM260_Result_Data_64_bytes_1[10];
	PlcInputs.ST40_1_DM260_Result_Data_64_bytes_1[11] := HwInputs.ST40_1_DM260_Result_Data_64_bytes_1[11];
	PlcInputs.ST40_1_DM260_Result_Data_64_bytes_1[12] := HwInputs.ST40_1_DM260_Result_Data_64_bytes_1[12];
	PlcInputs.ST40_1_DM260_Result_Data_64_bytes_1[13] := HwInputs.ST40_1_DM260_Result_Data_64_bytes_1[13];
	PlcInputs.ST40_1_DM260_Result_Data_64_bytes_1[14] := HwInputs.ST40_1_DM260_Result_Data_64_bytes_1[14];
	PlcInputs.ST40_1_DM260_Result_Data_64_bytes_1[15] := HwInputs.ST40_1_DM260_Result_Data_64_bytes_1[15];
	PlcInputs.ST40_1_DM260_Result_Data_64_bytes_1[16] := HwInputs.ST40_1_DM260_Result_Data_64_bytes_1[16];
	PlcInputs.ST40_1_DM260_Result_Data_64_bytes_1[17] := HwInputs.ST40_1_DM260_Result_Data_64_bytes_1[17];
	PlcInputs.ST40_1_DM260_Result_Data_64_bytes_1[18] := HwInputs.ST40_1_DM260_Result_Data_64_bytes_1[18];
	PlcInputs.ST40_1_DM260_Result_Data_64_bytes_1[19] := HwInputs.ST40_1_DM260_Result_Data_64_bytes_1[19];
	PlcInputs.ST40_1_DM260_Result_Data_64_bytes_1[20] := HwInputs.ST40_1_DM260_Result_Data_64_bytes_1[20];
	PlcInputs.ST40_1_DM260_Result_Data_64_bytes_1[21] := HwInputs.ST40_1_DM260_Result_Data_64_bytes_1[21];
	PlcInputs.ST40_1_DM260_Result_Data_64_bytes_1[22] := HwInputs.ST40_1_DM260_Result_Data_64_bytes_1[22];
	PlcInputs.ST40_1_DM260_Result_Data_64_bytes_1[23] := HwInputs.ST40_1_DM260_Result_Data_64_bytes_1[23];
	PlcInputs.ST40_1_DM260_Result_Data_64_bytes_1[24] := HwInputs.ST40_1_DM260_Result_Data_64_bytes_1[24];
	PlcInputs.ST40_1_DM260_Result_Data_64_bytes_1[25] := HwInputs.ST40_1_DM260_Result_Data_64_bytes_1[25];
	PlcInputs.ST40_1_DM260_Result_Data_64_bytes_1[26] := HwInputs.ST40_1_DM260_Result_Data_64_bytes_1[26];
	PlcInputs.ST40_1_DM260_Result_Data_64_bytes_1[27] := HwInputs.ST40_1_DM260_Result_Data_64_bytes_1[27];
	PlcInputs.ST40_1_DM260_Result_Data_64_bytes_1[28] := HwInputs.ST40_1_DM260_Result_Data_64_bytes_1[28];
	PlcInputs.ST40_1_DM260_Result_Data_64_bytes_1[29] := HwInputs.ST40_1_DM260_Result_Data_64_bytes_1[29];
	PlcInputs.ST40_1_DM260_Result_Data_64_bytes_1[30] := HwInputs.ST40_1_DM260_Result_Data_64_bytes_1[30];
	PlcInputs.ST40_1_DM260_Result_Data_64_bytes_1[31] := HwInputs.ST40_1_DM260_Result_Data_64_bytes_1[31];
	PlcInputs.ST40_1_DM260_Result_Data_64_bytes_1[32] := HwInputs.ST40_1_DM260_Result_Data_64_bytes_1[32];
	PlcInputs.ST40_1_DM260_Result_Data_64_bytes_1[33] := HwInputs.ST40_1_DM260_Result_Data_64_bytes_1[33];
	PlcInputs.ST40_1_DM260_Result_Data_64_bytes_1[34] := HwInputs.ST40_1_DM260_Result_Data_64_bytes_1[34];
	PlcInputs.ST40_1_DM260_Result_Data_64_bytes_1[35] := HwInputs.ST40_1_DM260_Result_Data_64_bytes_1[35];
	PlcInputs.ST40_1_DM260_Result_Data_64_bytes_1[36] := HwInputs.ST40_1_DM260_Result_Data_64_bytes_1[36];
	PlcInputs.ST40_1_DM260_Result_Data_64_bytes_1[37] := HwInputs.ST40_1_DM260_Result_Data_64_bytes_1[37];
	PlcInputs.ST40_1_DM260_Result_Data_64_bytes_1[38] := HwInputs.ST40_1_DM260_Result_Data_64_bytes_1[38];
	PlcInputs.ST40_1_DM260_Result_Data_64_bytes_1[39] := HwInputs.ST40_1_DM260_Result_Data_64_bytes_1[39];
	PlcInputs.ST40_1_DM260_Result_Data_64_bytes_1[40] := HwInputs.ST40_1_DM260_Result_Data_64_bytes_1[40];
	PlcInputs.ST40_1_DM260_Result_Data_64_bytes_1[41] := HwInputs.ST40_1_DM260_Result_Data_64_bytes_1[41];
	PlcInputs.ST40_1_DM260_Result_Data_64_bytes_1[42] := HwInputs.ST40_1_DM260_Result_Data_64_bytes_1[42];
	PlcInputs.ST40_1_DM260_Result_Data_64_bytes_1[43] := HwInputs.ST40_1_DM260_Result_Data_64_bytes_1[43];
	PlcInputs.ST40_1_DM260_Result_Data_64_bytes_1[44] := HwInputs.ST40_1_DM260_Result_Data_64_bytes_1[44];
	PlcInputs.ST40_1_DM260_Result_Data_64_bytes_1[45] := HwInputs.ST40_1_DM260_Result_Data_64_bytes_1[45];
	PlcInputs.ST40_1_DM260_Result_Data_64_bytes_1[46] := HwInputs.ST40_1_DM260_Result_Data_64_bytes_1[46];
	PlcInputs.ST40_1_DM260_Result_Data_64_bytes_1[47] := HwInputs.ST40_1_DM260_Result_Data_64_bytes_1[47];
	PlcInputs.ST40_1_DM260_Result_Data_64_bytes_1[48] := HwInputs.ST40_1_DM260_Result_Data_64_bytes_1[48];
	PlcInputs.ST40_1_DM260_Result_Data_64_bytes_1[49] := HwInputs.ST40_1_DM260_Result_Data_64_bytes_1[49];
	PlcInputs.ST40_1_DM260_Result_Data_64_bytes_1[50] := HwInputs.ST40_1_DM260_Result_Data_64_bytes_1[50];
	PlcInputs.ST40_1_DM260_Result_Data_64_bytes_1[51] := HwInputs.ST40_1_DM260_Result_Data_64_bytes_1[51];
	PlcInputs.ST40_1_DM260_Result_Data_64_bytes_1[52] := HwInputs.ST40_1_DM260_Result_Data_64_bytes_1[52];
	PlcInputs.ST40_1_DM260_Result_Data_64_bytes_1[53] := HwInputs.ST40_1_DM260_Result_Data_64_bytes_1[53];
	PlcInputs.ST40_1_DM260_Result_Data_64_bytes_1[54] := HwInputs.ST40_1_DM260_Result_Data_64_bytes_1[54];
	PlcInputs.ST40_1_DM260_Result_Data_64_bytes_1[55] := HwInputs.ST40_1_DM260_Result_Data_64_bytes_1[55];
	PlcInputs.ST40_1_DM260_Result_Data_64_bytes_1[56] := HwInputs.ST40_1_DM260_Result_Data_64_bytes_1[56];
	PlcInputs.ST40_1_DM260_Result_Data_64_bytes_1[57] := HwInputs.ST40_1_DM260_Result_Data_64_bytes_1[57];
	PlcInputs.ST40_1_DM260_Result_Data_64_bytes_1[58] := HwInputs.ST40_1_DM260_Result_Data_64_bytes_1[58];
	PlcInputs.ST40_1_DM260_Result_Data_64_bytes_1[59] := HwInputs.ST40_1_DM260_Result_Data_64_bytes_1[59];
	PlcInputs.ST40_1_DM260_Result_Data_64_bytes_1[60] := HwInputs.ST40_1_DM260_Result_Data_64_bytes_1[60];
	PlcInputs.ST40_1_DM260_Result_Data_64_bytes_1[61] := HwInputs.ST40_1_DM260_Result_Data_64_bytes_1[61];
	PlcInputs.ST40_1_DM260_Result_Data_64_bytes_1[62] := HwInputs.ST40_1_DM260_Result_Data_64_bytes_1[62];
	PlcInputs.ST40_1_DM260_Result_Data_64_bytes_1[63] := HwInputs.ST40_1_DM260_Result_Data_64_bytes_1[63];
	PlcInputs.ST40_1_DM260_Result_Data_64_bytes_1[64] := HwInputs.ST40_1_DM260_Result_Data_64_bytes_1[64];
	PlcInputs.ST40_1_DM260_Result_Data_64_bytes_1[65] := HwInputs.ST40_1_DM260_Result_Data_64_bytes_1[65];
	PlcInputs.ST40_1_DM260_Result_Data_64_bytes_1[66] := HwInputs.ST40_1_DM260_Result_Data_64_bytes_1[66];
	PlcInputs.ST40_1_DM260_Result_Data_64_bytes_1[67] := HwInputs.ST40_1_DM260_Result_Data_64_bytes_1[67];
	PlcInputs.ST40_1_DM260_Result_Data_64_bytes_1[68] := HwInputs.ST40_1_DM260_Result_Data_64_bytes_1[68];
	PlcInputs.ST40_1_DM260_Result_Data_64_bytes_1[69] := HwInputs.ST40_1_DM260_Result_Data_64_bytes_1[69];
	PlcInputs.ST40_1_DM260_Result_Data_64_bytes_1[70] := HwInputs.ST40_1_DM260_Result_Data_64_bytes_1[70];
	PlcInputs.ST40_1_DM260_Result_Data_64_bytes_1[71] := HwInputs.ST40_1_DM260_Result_Data_64_bytes_1[71];
	PlcInputs.ST40_2_Promess_Menu_30_01_In_1 := HwInputs.ST40_2_Promess_Menu_30_01_In_1;
	PlcInputs.ST40_2_Promess_Menu_30_02_In_1 := HwInputs.ST40_2_Promess_Menu_30_02_In_1;
	PlcInputs.ST40_2_Promess_Menu_30_03_In_1 := HwInputs.ST40_2_Promess_Menu_30_03_In_1;
	PlcInputs.ST40_2_Promess_Menu_30_04_In_1 := HwInputs.ST40_2_Promess_Menu_30_04_In_1;
	PlcInputs.ST40_2_Promess_Menu_30_05_In_1 := HwInputs.ST40_2_Promess_Menu_30_05_In_1;
	PlcInputs.ST40_2_Promess_Menu_30_06_In_1 := HwInputs.ST40_2_Promess_Menu_30_06_In_1;
	PlcInputs.ST40_2_Promess_Menu_30_07_In_1 := HwInputs.ST40_2_Promess_Menu_30_07_In_1;
	PlcInputs.ST40_2_Promess_Menu_30_08_In_1 := HwInputs.ST40_2_Promess_Menu_30_08_In_1;
	PlcInputs.ST40_2_Promess_Menu_30_09_In_1 := HwInputs.ST40_2_Promess_Menu_30_09_In_1;
	PlcInputs.ST40_2_Promess_Menu_30_10_In_1 := HwInputs.ST40_2_Promess_Menu_30_10_In_1;
	PlcInputs.ST40_2_Promess_Menu_30_11_In_1 := HwInputs.ST40_2_Promess_Menu_30_11_In_1;
	PlcInputs.ST40_2_Promess_Menu_30_12_In_1 := HwInputs.ST40_2_Promess_Menu_30_12_In_1;
	PlcInputs.ST40_2_Promess_Menu_30_13_In_1 := HwInputs.ST40_2_Promess_Menu_30_13_In_1;
	PlcInputs.ST40_2_Promess_Menu_30_14_In_1 := HwInputs.ST40_2_Promess_Menu_30_14_In_1;
	PlcInputs.ST40_2_Promess_Menu_30_15_In_1 := HwInputs.ST40_2_Promess_Menu_30_15_In_1;
	PlcInputs.ST40_2_Promess_Menu_30_16_In_1 := HwInputs.ST40_2_Promess_Menu_30_16_In_1;
	PlcInputs.ST40_2_Promess_Menu_30_17_In_1 := HwInputs.ST40_2_Promess_Menu_30_17_In_1;
	PlcInputs.ST40_2_Promess_Menu_30_18_In_1 := HwInputs.ST40_2_Promess_Menu_30_18_In_1;
	PlcInputs.ST40_2_Promess_Menu_30_19_In_1 := HwInputs.ST40_2_Promess_Menu_30_19_In_1;
	PlcInputs.ST40_2_Promess_Menu_30_20_In_1 := HwInputs.ST40_2_Promess_Menu_30_20_In_1;
	PlcInputs.ST40_2_Promess_Menu_30_21_In_1 := HwInputs.ST40_2_Promess_Menu_30_21_In_1;
	PlcInputs.ST40_2_Promess_Menu_30_22_In_1 := HwInputs.ST40_2_Promess_Menu_30_22_In_1;
	PlcInputs.ST40_2_Promess_Menu_30_23_In_1 := HwInputs.ST40_2_Promess_Menu_30_23_In_1;
	PlcInputs.ST40_2_Promess_Menu_30_24_In_1 := HwInputs.ST40_2_Promess_Menu_30_24_In_1;
	PlcInputs.ST40_2_Promess_Menu_30_25_In_1 := HwInputs.ST40_2_Promess_Menu_30_25_In_1;
	PlcInputs.ST40_2_Promess_Menu_30_26_In_1 := HwInputs.ST40_2_Promess_Menu_30_26_In_1;
	PlcInputs.ST40_2_Promess_Menu_30_27_In_1 := HwInputs.ST40_2_Promess_Menu_30_27_In_1;
	PlcInputs.ST40_2_Promess_Menu_30_28_In_1 := HwInputs.ST40_2_Promess_Menu_30_28_In_1;
	PlcInputs.ST40_2_Promess_Menu_30_29_In_1 := HwInputs.ST40_2_Promess_Menu_30_29_In_1;
	PlcInputs.ST40_2_Promess_Menu_30_30_In_1 := HwInputs.ST40_2_Promess_Menu_30_30_In_1;
	PlcInputs.ST40_2_Promess_Menu_30_31_In_1 := HwInputs.ST40_2_Promess_Menu_30_31_In_1;
	PlcInputs.ST40_2_Promess_Menu_30_32_In_1 := HwInputs.ST40_2_Promess_Menu_30_32_In_1;
	PlcInputs.ST40_ET200SP_CM_4xIO_Link_1[0] := HwInputs.ST40_ET200SP_CM_4xIO_Link_1[0];
	PlcInputs.ST40_ET200SP_CM_4xIO_Link_1[1] := HwInputs.ST40_ET200SP_CM_4xIO_Link_1[1];
	PlcInputs.ST40_ET200SP_CM_4xIO_Link_1[2] := HwInputs.ST40_ET200SP_CM_4xIO_Link_1[2];
	PlcInputs.ST40_ET200SP_CM_4xIO_Link_1[3] := HwInputs.ST40_ET200SP_CM_4xIO_Link_1[3];
	PlcInputs.ST40_ET200SP_CM_4xIO_Link_1[4] := HwInputs.ST40_ET200SP_CM_4xIO_Link_1[4];
	PlcInputs.ST40_ET200SP_CM_4xIO_Link_1[5] := HwInputs.ST40_ET200SP_CM_4xIO_Link_1[5];
	PlcInputs.ST40_ET200SP_CM_4xIO_Link_1[6] := HwInputs.ST40_ET200SP_CM_4xIO_Link_1[6];
	PlcInputs.ST40_ET200SP_CM_4xIO_Link_1[7] := HwInputs.ST40_ET200SP_CM_4xIO_Link_1[7];
	PlcInputs.ST40_ET200SP_CM_4xIO_Link_1[8] := HwInputs.ST40_ET200SP_CM_4xIO_Link_1[8];
	PlcInputs.ST40_ET200SP_CM_4xIO_Link_1[9] := HwInputs.ST40_ET200SP_CM_4xIO_Link_1[9];
	PlcInputs.ST40_ET200SP_CM_4xIO_Link_1[10] := HwInputs.ST40_ET200SP_CM_4xIO_Link_1[10];
	PlcInputs.ST40_ET200SP_CM_4xIO_Link_1[11] := HwInputs.ST40_ET200SP_CM_4xIO_Link_1[11];
	PlcInputs.ST40_ET200SP_CM_4xIO_Link_1[12] := HwInputs.ST40_ET200SP_CM_4xIO_Link_1[12];
	PlcInputs.ST40_ET200SP_CM_4xIO_Link_1[13] := HwInputs.ST40_ET200SP_CM_4xIO_Link_1[13];
	PlcInputs.ST40_ET200SP_CM_4xIO_Link_1[14] := HwInputs.ST40_ET200SP_CM_4xIO_Link_1[14];
	PlcInputs.ST40_ET200SP_CM_4xIO_Link_1[15] := HwInputs.ST40_ET200SP_CM_4xIO_Link_1[15];
	PlcInputs.ST40_ET200SP_CM_4xIO_Link_1[16] := HwInputs.ST40_ET200SP_CM_4xIO_Link_1[16];
	PlcInputs.ST40_ET200SP_CM_4xIO_Link_1[17] := HwInputs.ST40_ET200SP_CM_4xIO_Link_1[17];
	PlcInputs.ST40_ET200SP_CM_4xIO_Link_1[18] := HwInputs.ST40_ET200SP_CM_4xIO_Link_1[18];
	PlcInputs.ST40_ET200SP_CM_4xIO_Link_1[19] := HwInputs.ST40_ET200SP_CM_4xIO_Link_1[19];
	PlcInputs.ST40_ET200SP_CM_4xIO_Link_1[20] := HwInputs.ST40_ET200SP_CM_4xIO_Link_1[20];
	PlcInputs.ST40_ET200SP_CM_4xIO_Link_1[21] := HwInputs.ST40_ET200SP_CM_4xIO_Link_1[21];
	PlcInputs.ST40_ET200SP_CM_4xIO_Link_1[22] := HwInputs.ST40_ET200SP_CM_4xIO_Link_1[22];
	PlcInputs.ST40_ET200SP_CM_4xIO_Link_1[23] := HwInputs.ST40_ET200SP_CM_4xIO_Link_1[23];
	PlcInputs.ST40_ET200SP_CM_4xIO_Link_1[24] := HwInputs.ST40_ET200SP_CM_4xIO_Link_1[24];
	PlcInputs.ST40_ET200SP_CM_4xIO_Link_1[25] := HwInputs.ST40_ET200SP_CM_4xIO_Link_1[25];
	PlcInputs.ST40_ET200SP_CM_4xIO_Link_1[26] := HwInputs.ST40_ET200SP_CM_4xIO_Link_1[26];
	PlcInputs.ST40_ET200SP_CM_4xIO_Link_1[27] := HwInputs.ST40_ET200SP_CM_4xIO_Link_1[27];
	PlcInputs.ST40_ET200SP_CM_4xIO_Link_1[28] := HwInputs.ST40_ET200SP_CM_4xIO_Link_1[28];
	PlcInputs.ST40_ET200SP_CM_4xIO_Link_1[29] := HwInputs.ST40_ET200SP_CM_4xIO_Link_1[29];
	PlcInputs.ST40_ET200SP_CM_4xIO_Link_1[30] := HwInputs.ST40_ET200SP_CM_4xIO_Link_1[30];
	PlcInputs.ST40_ET200SP_CM_4xIO_Link_1[31] := HwInputs.ST40_ET200SP_CM_4xIO_Link_1[31];
	PlcInputs.ST40_ET200SP_CM_4xIO_Link_2[0] := HwInputs.ST40_ET200SP_CM_4xIO_Link_2[0];
	PlcInputs.ST40_ET200SP_CM_4xIO_Link_2[1] := HwInputs.ST40_ET200SP_CM_4xIO_Link_2[1];
	PlcInputs.ST40_ET200SP_CM_4xIO_Link_2[2] := HwInputs.ST40_ET200SP_CM_4xIO_Link_2[2];
	PlcInputs.ST40_ET200SP_CM_4xIO_Link_2[3] := HwInputs.ST40_ET200SP_CM_4xIO_Link_2[3];
	PlcInputs.ST40_ET200SP_CM_4xIO_Link_2[4] := HwInputs.ST40_ET200SP_CM_4xIO_Link_2[4];
	PlcInputs.ST40_ET200SP_CM_4xIO_Link_2[5] := HwInputs.ST40_ET200SP_CM_4xIO_Link_2[5];
	PlcInputs.ST40_ET200SP_CM_4xIO_Link_2[6] := HwInputs.ST40_ET200SP_CM_4xIO_Link_2[6];
	PlcInputs.ST40_ET200SP_CM_4xIO_Link_2[7] := HwInputs.ST40_ET200SP_CM_4xIO_Link_2[7];
	PlcInputs.ST40_ET200SP_CM_4xIO_Link_2[8] := HwInputs.ST40_ET200SP_CM_4xIO_Link_2[8];
	PlcInputs.ST40_ET200SP_CM_4xIO_Link_2[9] := HwInputs.ST40_ET200SP_CM_4xIO_Link_2[9];
	PlcInputs.ST40_ET200SP_CM_4xIO_Link_2[10] := HwInputs.ST40_ET200SP_CM_4xIO_Link_2[10];
	PlcInputs.ST40_ET200SP_CM_4xIO_Link_2[11] := HwInputs.ST40_ET200SP_CM_4xIO_Link_2[11];
	PlcInputs.ST40_ET200SP_CM_4xIO_Link_2[12] := HwInputs.ST40_ET200SP_CM_4xIO_Link_2[12];
	PlcInputs.ST40_ET200SP_CM_4xIO_Link_2[13] := HwInputs.ST40_ET200SP_CM_4xIO_Link_2[13];
	PlcInputs.ST40_ET200SP_CM_4xIO_Link_2[14] := HwInputs.ST40_ET200SP_CM_4xIO_Link_2[14];
	PlcInputs.ST40_ET200SP_CM_4xIO_Link_2[15] := HwInputs.ST40_ET200SP_CM_4xIO_Link_2[15];
	PlcInputs.ST40_ET200SP_CM_4xIO_Link_2[16] := HwInputs.ST40_ET200SP_CM_4xIO_Link_2[16];
	PlcInputs.ST40_ET200SP_CM_4xIO_Link_2[17] := HwInputs.ST40_ET200SP_CM_4xIO_Link_2[17];
	PlcInputs.ST40_ET200SP_CM_4xIO_Link_2[18] := HwInputs.ST40_ET200SP_CM_4xIO_Link_2[18];
	PlcInputs.ST40_ET200SP_CM_4xIO_Link_2[19] := HwInputs.ST40_ET200SP_CM_4xIO_Link_2[19];
	PlcInputs.ST40_ET200SP_CM_4xIO_Link_2[20] := HwInputs.ST40_ET200SP_CM_4xIO_Link_2[20];
	PlcInputs.ST40_ET200SP_CM_4xIO_Link_2[21] := HwInputs.ST40_ET200SP_CM_4xIO_Link_2[21];
	PlcInputs.ST40_ET200SP_CM_4xIO_Link_2[22] := HwInputs.ST40_ET200SP_CM_4xIO_Link_2[22];
	PlcInputs.ST40_ET200SP_CM_4xIO_Link_2[23] := HwInputs.ST40_ET200SP_CM_4xIO_Link_2[23];
	PlcInputs.ST40_ET200SP_CM_4xIO_Link_2[24] := HwInputs.ST40_ET200SP_CM_4xIO_Link_2[24];
	PlcInputs.ST40_ET200SP_CM_4xIO_Link_2[25] := HwInputs.ST40_ET200SP_CM_4xIO_Link_2[25];
	PlcInputs.ST40_ET200SP_CM_4xIO_Link_2[26] := HwInputs.ST40_ET200SP_CM_4xIO_Link_2[26];
	PlcInputs.ST40_ET200SP_CM_4xIO_Link_2[27] := HwInputs.ST40_ET200SP_CM_4xIO_Link_2[27];
	PlcInputs.ST40_ET200SP_CM_4xIO_Link_2[28] := HwInputs.ST40_ET200SP_CM_4xIO_Link_2[28];
	PlcInputs.ST40_ET200SP_CM_4xIO_Link_2[29] := HwInputs.ST40_ET200SP_CM_4xIO_Link_2[29];
	PlcInputs.ST40_ET200SP_CM_4xIO_Link_2[30] := HwInputs.ST40_ET200SP_CM_4xIO_Link_2[30];
	PlcInputs.ST40_ET200SP_CM_4xIO_Link_2[31] := HwInputs.ST40_ET200SP_CM_4xIO_Link_2[31];
	PlcInputs.ST40_ET200SP_DI_8x24VDC_ST_1 := HwInputs.ST40_ET200SP_DI_8x24VDC_ST_1;
	PlcInputs.ST40_ET200SP_DI_8x24VDC_ST_2 := HwInputs.ST40_ET200SP_DI_8x24VDC_ST_2;
	PlcInputs.ST40_ET200SP_DI_16x24VDC_ST_1 := HwInputs.ST40_ET200SP_DI_16x24VDC_ST_1;
	PlcInputs.ST40_ET200SP_DI_8x24VDC_ST_3 := HwInputs.ST40_ET200SP_DI_8x24VDC_ST_3;
END_FUNCTION

(* ---- CopyOutputs.st ---- *)
FUNCTION CopyOutputs
	VAR_EXTERNAL
		HwOutputs : HwOutputs;
		PlcOutputs : PlcOutputs;
	END_VAR
	HwOutputs.ST40_2_DM260_Acquisition_Control_1 := PlcOutputs.ST40_2_DM260_Acquisition_Control_1;
	HwOutputs.ST40_2_DM260_Results_Control_1 := PlcOutputs.ST40_2_DM260_Results_Control_1;
	HwOutputs.ST40_2_DM260_Soft_Event_Control_1 := PlcOutputs.ST40_2_DM260_Soft_Event_Control_1;
	HwOutputs.ST40_2_DM260_User_Data_64_bytes_1[0] := PlcOutputs.ST40_2_DM260_User_Data_64_bytes_1[0];
	HwOutputs.ST40_2_DM260_User_Data_64_bytes_1[1] := PlcOutputs.ST40_2_DM260_User_Data_64_bytes_1[1];
	HwOutputs.ST40_2_DM260_User_Data_64_bytes_1[2] := PlcOutputs.ST40_2_DM260_User_Data_64_bytes_1[2];
	HwOutputs.ST40_2_DM260_User_Data_64_bytes_1[3] := PlcOutputs.ST40_2_DM260_User_Data_64_bytes_1[3];
	HwOutputs.ST40_2_DM260_User_Data_64_bytes_1[4] := PlcOutputs.ST40_2_DM260_User_Data_64_bytes_1[4];
	HwOutputs.ST40_2_DM260_User_Data_64_bytes_1[5] := PlcOutputs.ST40_2_DM260_User_Data_64_bytes_1[5];
	HwOutputs.ST40_2_DM260_User_Data_64_bytes_1[6] := PlcOutputs.ST40_2_DM260_User_Data_64_bytes_1[6];
	HwOutputs.ST40_2_DM260_User_Data_64_bytes_1[7] := PlcOutputs.ST40_2_DM260_User_Data_64_bytes_1[7];
	HwOutputs.ST40_2_DM260_User_Data_64_bytes_1[8] := PlcOutputs.ST40_2_DM260_User_Data_64_bytes_1[8];
	HwOutputs.ST40_2_DM260_User_Data_64_bytes_1[9] := PlcOutputs.ST40_2_DM260_User_Data_64_bytes_1[9];
	HwOutputs.ST40_2_DM260_User_Data_64_bytes_1[10] := PlcOutputs.ST40_2_DM260_User_Data_64_bytes_1[10];
	HwOutputs.ST40_2_DM260_User_Data_64_bytes_1[11] := PlcOutputs.ST40_2_DM260_User_Data_64_bytes_1[11];
	HwOutputs.ST40_2_DM260_User_Data_64_bytes_1[12] := PlcOutputs.ST40_2_DM260_User_Data_64_bytes_1[12];
	HwOutputs.ST40_2_DM260_User_Data_64_bytes_1[13] := PlcOutputs.ST40_2_DM260_User_Data_64_bytes_1[13];
	HwOutputs.ST40_2_DM260_User_Data_64_bytes_1[14] := PlcOutputs.ST40_2_DM260_User_Data_64_bytes_1[14];
	HwOutputs.ST40_2_DM260_User_Data_64_bytes_1[15] := PlcOutputs.ST40_2_DM260_User_Data_64_bytes_1[15];
	HwOutputs.ST40_2_DM260_User_Data_64_bytes_1[16] := PlcOutputs.ST40_2_DM260_User_Data_64_bytes_1[16];
	HwOutputs.ST40_2_DM260_User_Data_64_bytes_1[17] := PlcOutputs.ST40_2_DM260_User_Data_64_bytes_1[17];
	HwOutputs.ST40_2_DM260_User_Data_64_bytes_1[18] := PlcOutputs.ST40_2_DM260_User_Data_64_bytes_1[18];
	HwOutputs.ST40_2_DM260_User_Data_64_bytes_1[19] := PlcOutputs.ST40_2_DM260_User_Data_64_bytes_1[19];
	HwOutputs.ST40_2_DM260_User_Data_64_bytes_1[20] := PlcOutputs.ST40_2_DM260_User_Data_64_bytes_1[20];
	HwOutputs.ST40_2_DM260_User_Data_64_bytes_1[21] := PlcOutputs.ST40_2_DM260_User_Data_64_bytes_1[21];
	HwOutputs.ST40_2_DM260_User_Data_64_bytes_1[22] := PlcOutputs.ST40_2_DM260_User_Data_64_bytes_1[22];
	HwOutputs.ST40_2_DM260_User_Data_64_bytes_1[23] := PlcOutputs.ST40_2_DM260_User_Data_64_bytes_1[23];
	HwOutputs.ST40_2_DM260_User_Data_64_bytes_1[24] := PlcOutputs.ST40_2_DM260_User_Data_64_bytes_1[24];
	HwOutputs.ST40_2_DM260_User_Data_64_bytes_1[25] := PlcOutputs.ST40_2_DM260_User_Data_64_bytes_1[25];
	HwOutputs.ST40_2_DM260_User_Data_64_bytes_1[26] := PlcOutputs.ST40_2_DM260_User_Data_64_bytes_1[26];
	HwOutputs.ST40_2_DM260_User_Data_64_bytes_1[27] := PlcOutputs.ST40_2_DM260_User_Data_64_bytes_1[27];
	HwOutputs.ST40_2_DM260_User_Data_64_bytes_1[28] := PlcOutputs.ST40_2_DM260_User_Data_64_bytes_1[28];
	HwOutputs.ST40_2_DM260_User_Data_64_bytes_1[29] := PlcOutputs.ST40_2_DM260_User_Data_64_bytes_1[29];
	HwOutputs.ST40_2_DM260_User_Data_64_bytes_1[30] := PlcOutputs.ST40_2_DM260_User_Data_64_bytes_1[30];
	HwOutputs.ST40_2_DM260_User_Data_64_bytes_1[31] := PlcOutputs.ST40_2_DM260_User_Data_64_bytes_1[31];
	HwOutputs.ST40_2_DM260_User_Data_64_bytes_1[32] := PlcOutputs.ST40_2_DM260_User_Data_64_bytes_1[32];
	HwOutputs.ST40_2_DM260_User_Data_64_bytes_1[33] := PlcOutputs.ST40_2_DM260_User_Data_64_bytes_1[33];
	HwOutputs.ST40_2_DM260_User_Data_64_bytes_1[34] := PlcOutputs.ST40_2_DM260_User_Data_64_bytes_1[34];
	HwOutputs.ST40_2_DM260_User_Data_64_bytes_1[35] := PlcOutputs.ST40_2_DM260_User_Data_64_bytes_1[35];
	HwOutputs.ST40_2_DM260_User_Data_64_bytes_1[36] := PlcOutputs.ST40_2_DM260_User_Data_64_bytes_1[36];
	HwOutputs.ST40_2_DM260_User_Data_64_bytes_1[37] := PlcOutputs.ST40_2_DM260_User_Data_64_bytes_1[37];
	HwOutputs.ST40_2_DM260_User_Data_64_bytes_1[38] := PlcOutputs.ST40_2_DM260_User_Data_64_bytes_1[38];
	HwOutputs.ST40_2_DM260_User_Data_64_bytes_1[39] := PlcOutputs.ST40_2_DM260_User_Data_64_bytes_1[39];
	HwOutputs.ST40_2_DM260_User_Data_64_bytes_1[40] := PlcOutputs.ST40_2_DM260_User_Data_64_bytes_1[40];
	HwOutputs.ST40_2_DM260_User_Data_64_bytes_1[41] := PlcOutputs.ST40_2_DM260_User_Data_64_bytes_1[41];
	HwOutputs.ST40_2_DM260_User_Data_64_bytes_1[42] := PlcOutputs.ST40_2_DM260_User_Data_64_bytes_1[42];
	HwOutputs.ST40_2_DM260_User_Data_64_bytes_1[43] := PlcOutputs.ST40_2_DM260_User_Data_64_bytes_1[43];
	HwOutputs.ST40_2_DM260_User_Data_64_bytes_1[44] := PlcOutputs.ST40_2_DM260_User_Data_64_bytes_1[44];
	HwOutputs.ST40_2_DM260_User_Data_64_bytes_1[45] := PlcOutputs.ST40_2_DM260_User_Data_64_bytes_1[45];
	HwOutputs.ST40_2_DM260_User_Data_64_bytes_1[46] := PlcOutputs.ST40_2_DM260_User_Data_64_bytes_1[46];
	HwOutputs.ST40_2_DM260_User_Data_64_bytes_1[47] := PlcOutputs.ST40_2_DM260_User_Data_64_bytes_1[47];
	HwOutputs.ST40_2_DM260_User_Data_64_bytes_1[48] := PlcOutputs.ST40_2_DM260_User_Data_64_bytes_1[48];
	HwOutputs.ST40_2_DM260_User_Data_64_bytes_1[49] := PlcOutputs.ST40_2_DM260_User_Data_64_bytes_1[49];
	HwOutputs.ST40_2_DM260_User_Data_64_bytes_1[50] := PlcOutputs.ST40_2_DM260_User_Data_64_bytes_1[50];
	HwOutputs.ST40_2_DM260_User_Data_64_bytes_1[51] := PlcOutputs.ST40_2_DM260_User_Data_64_bytes_1[51];
	HwOutputs.ST40_2_DM260_User_Data_64_bytes_1[52] := PlcOutputs.ST40_2_DM260_User_Data_64_bytes_1[52];
	HwOutputs.ST40_2_DM260_User_Data_64_bytes_1[53] := PlcOutputs.ST40_2_DM260_User_Data_64_bytes_1[53];
	HwOutputs.ST40_2_DM260_User_Data_64_bytes_1[54] := PlcOutputs.ST40_2_DM260_User_Data_64_bytes_1[54];
	HwOutputs.ST40_2_DM260_User_Data_64_bytes_1[55] := PlcOutputs.ST40_2_DM260_User_Data_64_bytes_1[55];
	HwOutputs.ST40_2_DM260_User_Data_64_bytes_1[56] := PlcOutputs.ST40_2_DM260_User_Data_64_bytes_1[56];
	HwOutputs.ST40_2_DM260_User_Data_64_bytes_1[57] := PlcOutputs.ST40_2_DM260_User_Data_64_bytes_1[57];
	HwOutputs.ST40_2_DM260_User_Data_64_bytes_1[58] := PlcOutputs.ST40_2_DM260_User_Data_64_bytes_1[58];
	HwOutputs.ST40_2_DM260_User_Data_64_bytes_1[59] := PlcOutputs.ST40_2_DM260_User_Data_64_bytes_1[59];
	HwOutputs.ST40_2_DM260_User_Data_64_bytes_1[60] := PlcOutputs.ST40_2_DM260_User_Data_64_bytes_1[60];
	HwOutputs.ST40_2_DM260_User_Data_64_bytes_1[61] := PlcOutputs.ST40_2_DM260_User_Data_64_bytes_1[61];
	HwOutputs.ST40_2_DM260_User_Data_64_bytes_1[62] := PlcOutputs.ST40_2_DM260_User_Data_64_bytes_1[62];
	HwOutputs.ST40_2_DM260_User_Data_64_bytes_1[63] := PlcOutputs.ST40_2_DM260_User_Data_64_bytes_1[63];
	HwOutputs.ST40_2_DM260_User_Data_64_bytes_1[64] := PlcOutputs.ST40_2_DM260_User_Data_64_bytes_1[64];
	HwOutputs.ST40_2_DM260_User_Data_64_bytes_1[65] := PlcOutputs.ST40_2_DM260_User_Data_64_bytes_1[65];
	HwOutputs.ST40_2_DM260_User_Data_64_bytes_1[66] := PlcOutputs.ST40_2_DM260_User_Data_64_bytes_1[66];
	HwOutputs.ST40_2_DM260_User_Data_64_bytes_1[67] := PlcOutputs.ST40_2_DM260_User_Data_64_bytes_1[67];
	HwOutputs.ST40_3_DM260_Acquisition_Control_1 := PlcOutputs.ST40_3_DM260_Acquisition_Control_1;
	HwOutputs.ST40_3_DM260_Results_Control_1 := PlcOutputs.ST40_3_DM260_Results_Control_1;
	HwOutputs.ST40_3_DM260_Soft_Event_Control_1 := PlcOutputs.ST40_3_DM260_Soft_Event_Control_1;
	HwOutputs.ST40_3_DM260_User_Data_64_bytes_1[0] := PlcOutputs.ST40_3_DM260_User_Data_64_bytes_1[0];
	HwOutputs.ST40_3_DM260_User_Data_64_bytes_1[1] := PlcOutputs.ST40_3_DM260_User_Data_64_bytes_1[1];
	HwOutputs.ST40_3_DM260_User_Data_64_bytes_1[2] := PlcOutputs.ST40_3_DM260_User_Data_64_bytes_1[2];
	HwOutputs.ST40_3_DM260_User_Data_64_bytes_1[3] := PlcOutputs.ST40_3_DM260_User_Data_64_bytes_1[3];
	HwOutputs.ST40_3_DM260_User_Data_64_bytes_1[4] := PlcOutputs.ST40_3_DM260_User_Data_64_bytes_1[4];
	HwOutputs.ST40_3_DM260_User_Data_64_bytes_1[5] := PlcOutputs.ST40_3_DM260_User_Data_64_bytes_1[5];
	HwOutputs.ST40_3_DM260_User_Data_64_bytes_1[6] := PlcOutputs.ST40_3_DM260_User_Data_64_bytes_1[6];
	HwOutputs.ST40_3_DM260_User_Data_64_bytes_1[7] := PlcOutputs.ST40_3_DM260_User_Data_64_bytes_1[7];
	HwOutputs.ST40_3_DM260_User_Data_64_bytes_1[8] := PlcOutputs.ST40_3_DM260_User_Data_64_bytes_1[8];
	HwOutputs.ST40_3_DM260_User_Data_64_bytes_1[9] := PlcOutputs.ST40_3_DM260_User_Data_64_bytes_1[9];
	HwOutputs.ST40_3_DM260_User_Data_64_bytes_1[10] := PlcOutputs.ST40_3_DM260_User_Data_64_bytes_1[10];
	HwOutputs.ST40_3_DM260_User_Data_64_bytes_1[11] := PlcOutputs.ST40_3_DM260_User_Data_64_bytes_1[11];
	HwOutputs.ST40_3_DM260_User_Data_64_bytes_1[12] := PlcOutputs.ST40_3_DM260_User_Data_64_bytes_1[12];
	HwOutputs.ST40_3_DM260_User_Data_64_bytes_1[13] := PlcOutputs.ST40_3_DM260_User_Data_64_bytes_1[13];
	HwOutputs.ST40_3_DM260_User_Data_64_bytes_1[14] := PlcOutputs.ST40_3_DM260_User_Data_64_bytes_1[14];
	HwOutputs.ST40_3_DM260_User_Data_64_bytes_1[15] := PlcOutputs.ST40_3_DM260_User_Data_64_bytes_1[15];
	HwOutputs.ST40_3_DM260_User_Data_64_bytes_1[16] := PlcOutputs.ST40_3_DM260_User_Data_64_bytes_1[16];
	HwOutputs.ST40_3_DM260_User_Data_64_bytes_1[17] := PlcOutputs.ST40_3_DM260_User_Data_64_bytes_1[17];
	HwOutputs.ST40_3_DM260_User_Data_64_bytes_1[18] := PlcOutputs.ST40_3_DM260_User_Data_64_bytes_1[18];
	HwOutputs.ST40_3_DM260_User_Data_64_bytes_1[19] := PlcOutputs.ST40_3_DM260_User_Data_64_bytes_1[19];
	HwOutputs.ST40_3_DM260_User_Data_64_bytes_1[20] := PlcOutputs.ST40_3_DM260_User_Data_64_bytes_1[20];
	HwOutputs.ST40_3_DM260_User_Data_64_bytes_1[21] := PlcOutputs.ST40_3_DM260_User_Data_64_bytes_1[21];
	HwOutputs.ST40_3_DM260_User_Data_64_bytes_1[22] := PlcOutputs.ST40_3_DM260_User_Data_64_bytes_1[22];
	HwOutputs.ST40_3_DM260_User_Data_64_bytes_1[23] := PlcOutputs.ST40_3_DM260_User_Data_64_bytes_1[23];
	HwOutputs.ST40_3_DM260_User_Data_64_bytes_1[24] := PlcOutputs.ST40_3_DM260_User_Data_64_bytes_1[24];
	HwOutputs.ST40_3_DM260_User_Data_64_bytes_1[25] := PlcOutputs.ST40_3_DM260_User_Data_64_bytes_1[25];
	HwOutputs.ST40_3_DM260_User_Data_64_bytes_1[26] := PlcOutputs.ST40_3_DM260_User_Data_64_bytes_1[26];
	HwOutputs.ST40_3_DM260_User_Data_64_bytes_1[27] := PlcOutputs.ST40_3_DM260_User_Data_64_bytes_1[27];
	HwOutputs.ST40_3_DM260_User_Data_64_bytes_1[28] := PlcOutputs.ST40_3_DM260_User_Data_64_bytes_1[28];
	HwOutputs.ST40_3_DM260_User_Data_64_bytes_1[29] := PlcOutputs.ST40_3_DM260_User_Data_64_bytes_1[29];
	HwOutputs.ST40_3_DM260_User_Data_64_bytes_1[30] := PlcOutputs.ST40_3_DM260_User_Data_64_bytes_1[30];
	HwOutputs.ST40_3_DM260_User_Data_64_bytes_1[31] := PlcOutputs.ST40_3_DM260_User_Data_64_bytes_1[31];
	HwOutputs.ST40_3_DM260_User_Data_64_bytes_1[32] := PlcOutputs.ST40_3_DM260_User_Data_64_bytes_1[32];
	HwOutputs.ST40_3_DM260_User_Data_64_bytes_1[33] := PlcOutputs.ST40_3_DM260_User_Data_64_bytes_1[33];
	HwOutputs.ST40_3_DM260_User_Data_64_bytes_1[34] := PlcOutputs.ST40_3_DM260_User_Data_64_bytes_1[34];
	HwOutputs.ST40_3_DM260_User_Data_64_bytes_1[35] := PlcOutputs.ST40_3_DM260_User_Data_64_bytes_1[35];
	HwOutputs.ST40_3_DM260_User_Data_64_bytes_1[36] := PlcOutputs.ST40_3_DM260_User_Data_64_bytes_1[36];
	HwOutputs.ST40_3_DM260_User_Data_64_bytes_1[37] := PlcOutputs.ST40_3_DM260_User_Data_64_bytes_1[37];
	HwOutputs.ST40_3_DM260_User_Data_64_bytes_1[38] := PlcOutputs.ST40_3_DM260_User_Data_64_bytes_1[38];
	HwOutputs.ST40_3_DM260_User_Data_64_bytes_1[39] := PlcOutputs.ST40_3_DM260_User_Data_64_bytes_1[39];
	HwOutputs.ST40_3_DM260_User_Data_64_bytes_1[40] := PlcOutputs.ST40_3_DM260_User_Data_64_bytes_1[40];
	HwOutputs.ST40_3_DM260_User_Data_64_bytes_1[41] := PlcOutputs.ST40_3_DM260_User_Data_64_bytes_1[41];
	HwOutputs.ST40_3_DM260_User_Data_64_bytes_1[42] := PlcOutputs.ST40_3_DM260_User_Data_64_bytes_1[42];
	HwOutputs.ST40_3_DM260_User_Data_64_bytes_1[43] := PlcOutputs.ST40_3_DM260_User_Data_64_bytes_1[43];
	HwOutputs.ST40_3_DM260_User_Data_64_bytes_1[44] := PlcOutputs.ST40_3_DM260_User_Data_64_bytes_1[44];
	HwOutputs.ST40_3_DM260_User_Data_64_bytes_1[45] := PlcOutputs.ST40_3_DM260_User_Data_64_bytes_1[45];
	HwOutputs.ST40_3_DM260_User_Data_64_bytes_1[46] := PlcOutputs.ST40_3_DM260_User_Data_64_bytes_1[46];
	HwOutputs.ST40_3_DM260_User_Data_64_bytes_1[47] := PlcOutputs.ST40_3_DM260_User_Data_64_bytes_1[47];
	HwOutputs.ST40_3_DM260_User_Data_64_bytes_1[48] := PlcOutputs.ST40_3_DM260_User_Data_64_bytes_1[48];
	HwOutputs.ST40_3_DM260_User_Data_64_bytes_1[49] := PlcOutputs.ST40_3_DM260_User_Data_64_bytes_1[49];
	HwOutputs.ST40_3_DM260_User_Data_64_bytes_1[50] := PlcOutputs.ST40_3_DM260_User_Data_64_bytes_1[50];
	HwOutputs.ST40_3_DM260_User_Data_64_bytes_1[51] := PlcOutputs.ST40_3_DM260_User_Data_64_bytes_1[51];
	HwOutputs.ST40_3_DM260_User_Data_64_bytes_1[52] := PlcOutputs.ST40_3_DM260_User_Data_64_bytes_1[52];
	HwOutputs.ST40_3_DM260_User_Data_64_bytes_1[53] := PlcOutputs.ST40_3_DM260_User_Data_64_bytes_1[53];
	HwOutputs.ST40_3_DM260_User_Data_64_bytes_1[54] := PlcOutputs.ST40_3_DM260_User_Data_64_bytes_1[54];
	HwOutputs.ST40_3_DM260_User_Data_64_bytes_1[55] := PlcOutputs.ST40_3_DM260_User_Data_64_bytes_1[55];
	HwOutputs.ST40_3_DM260_User_Data_64_bytes_1[56] := PlcOutputs.ST40_3_DM260_User_Data_64_bytes_1[56];
	HwOutputs.ST40_3_DM260_User_Data_64_bytes_1[57] := PlcOutputs.ST40_3_DM260_User_Data_64_bytes_1[57];
	HwOutputs.ST40_3_DM260_User_Data_64_bytes_1[58] := PlcOutputs.ST40_3_DM260_User_Data_64_bytes_1[58];
	HwOutputs.ST40_3_DM260_User_Data_64_bytes_1[59] := PlcOutputs.ST40_3_DM260_User_Data_64_bytes_1[59];
	HwOutputs.ST40_3_DM260_User_Data_64_bytes_1[60] := PlcOutputs.ST40_3_DM260_User_Data_64_bytes_1[60];
	HwOutputs.ST40_3_DM260_User_Data_64_bytes_1[61] := PlcOutputs.ST40_3_DM260_User_Data_64_bytes_1[61];
	HwOutputs.ST40_3_DM260_User_Data_64_bytes_1[62] := PlcOutputs.ST40_3_DM260_User_Data_64_bytes_1[62];
	HwOutputs.ST40_3_DM260_User_Data_64_bytes_1[63] := PlcOutputs.ST40_3_DM260_User_Data_64_bytes_1[63];
	HwOutputs.ST40_3_DM260_User_Data_64_bytes_1[64] := PlcOutputs.ST40_3_DM260_User_Data_64_bytes_1[64];
	HwOutputs.ST40_3_DM260_User_Data_64_bytes_1[65] := PlcOutputs.ST40_3_DM260_User_Data_64_bytes_1[65];
	HwOutputs.ST40_3_DM260_User_Data_64_bytes_1[66] := PlcOutputs.ST40_3_DM260_User_Data_64_bytes_1[66];
	HwOutputs.ST40_3_DM260_User_Data_64_bytes_1[67] := PlcOutputs.ST40_3_DM260_User_Data_64_bytes_1[67];
	HwOutputs.ST40_1_DM260_Acquisition_Control_1 := PlcOutputs.ST40_1_DM260_Acquisition_Control_1;
	HwOutputs.ST40_1_DM260_Results_Control_1 := PlcOutputs.ST40_1_DM260_Results_Control_1;
	HwOutputs.ST40_1_DM260_Soft_Event_Control_1 := PlcOutputs.ST40_1_DM260_Soft_Event_Control_1;
	HwOutputs.ST40_1_DM260_User_Data_64_bytes_1[0] := PlcOutputs.ST40_1_DM260_User_Data_64_bytes_1[0];
	HwOutputs.ST40_1_DM260_User_Data_64_bytes_1[1] := PlcOutputs.ST40_1_DM260_User_Data_64_bytes_1[1];
	HwOutputs.ST40_1_DM260_User_Data_64_bytes_1[2] := PlcOutputs.ST40_1_DM260_User_Data_64_bytes_1[2];
	HwOutputs.ST40_1_DM260_User_Data_64_bytes_1[3] := PlcOutputs.ST40_1_DM260_User_Data_64_bytes_1[3];
	HwOutputs.ST40_1_DM260_User_Data_64_bytes_1[4] := PlcOutputs.ST40_1_DM260_User_Data_64_bytes_1[4];
	HwOutputs.ST40_1_DM260_User_Data_64_bytes_1[5] := PlcOutputs.ST40_1_DM260_User_Data_64_bytes_1[5];
	HwOutputs.ST40_1_DM260_User_Data_64_bytes_1[6] := PlcOutputs.ST40_1_DM260_User_Data_64_bytes_1[6];
	HwOutputs.ST40_1_DM260_User_Data_64_bytes_1[7] := PlcOutputs.ST40_1_DM260_User_Data_64_bytes_1[7];
	HwOutputs.ST40_1_DM260_User_Data_64_bytes_1[8] := PlcOutputs.ST40_1_DM260_User_Data_64_bytes_1[8];
	HwOutputs.ST40_1_DM260_User_Data_64_bytes_1[9] := PlcOutputs.ST40_1_DM260_User_Data_64_bytes_1[9];
	HwOutputs.ST40_1_DM260_User_Data_64_bytes_1[10] := PlcOutputs.ST40_1_DM260_User_Data_64_bytes_1[10];
	HwOutputs.ST40_1_DM260_User_Data_64_bytes_1[11] := PlcOutputs.ST40_1_DM260_User_Data_64_bytes_1[11];
	HwOutputs.ST40_1_DM260_User_Data_64_bytes_1[12] := PlcOutputs.ST40_1_DM260_User_Data_64_bytes_1[12];
	HwOutputs.ST40_1_DM260_User_Data_64_bytes_1[13] := PlcOutputs.ST40_1_DM260_User_Data_64_bytes_1[13];
	HwOutputs.ST40_1_DM260_User_Data_64_bytes_1[14] := PlcOutputs.ST40_1_DM260_User_Data_64_bytes_1[14];
	HwOutputs.ST40_1_DM260_User_Data_64_bytes_1[15] := PlcOutputs.ST40_1_DM260_User_Data_64_bytes_1[15];
	HwOutputs.ST40_1_DM260_User_Data_64_bytes_1[16] := PlcOutputs.ST40_1_DM260_User_Data_64_bytes_1[16];
	HwOutputs.ST40_1_DM260_User_Data_64_bytes_1[17] := PlcOutputs.ST40_1_DM260_User_Data_64_bytes_1[17];
	HwOutputs.ST40_1_DM260_User_Data_64_bytes_1[18] := PlcOutputs.ST40_1_DM260_User_Data_64_bytes_1[18];
	HwOutputs.ST40_1_DM260_User_Data_64_bytes_1[19] := PlcOutputs.ST40_1_DM260_User_Data_64_bytes_1[19];
	HwOutputs.ST40_1_DM260_User_Data_64_bytes_1[20] := PlcOutputs.ST40_1_DM260_User_Data_64_bytes_1[20];
	HwOutputs.ST40_1_DM260_User_Data_64_bytes_1[21] := PlcOutputs.ST40_1_DM260_User_Data_64_bytes_1[21];
	HwOutputs.ST40_1_DM260_User_Data_64_bytes_1[22] := PlcOutputs.ST40_1_DM260_User_Data_64_bytes_1[22];
	HwOutputs.ST40_1_DM260_User_Data_64_bytes_1[23] := PlcOutputs.ST40_1_DM260_User_Data_64_bytes_1[23];
	HwOutputs.ST40_1_DM260_User_Data_64_bytes_1[24] := PlcOutputs.ST40_1_DM260_User_Data_64_bytes_1[24];
	HwOutputs.ST40_1_DM260_User_Data_64_bytes_1[25] := PlcOutputs.ST40_1_DM260_User_Data_64_bytes_1[25];
	HwOutputs.ST40_1_DM260_User_Data_64_bytes_1[26] := PlcOutputs.ST40_1_DM260_User_Data_64_bytes_1[26];
	HwOutputs.ST40_1_DM260_User_Data_64_bytes_1[27] := PlcOutputs.ST40_1_DM260_User_Data_64_bytes_1[27];
	HwOutputs.ST40_1_DM260_User_Data_64_bytes_1[28] := PlcOutputs.ST40_1_DM260_User_Data_64_bytes_1[28];
	HwOutputs.ST40_1_DM260_User_Data_64_bytes_1[29] := PlcOutputs.ST40_1_DM260_User_Data_64_bytes_1[29];
	HwOutputs.ST40_1_DM260_User_Data_64_bytes_1[30] := PlcOutputs.ST40_1_DM260_User_Data_64_bytes_1[30];
	HwOutputs.ST40_1_DM260_User_Data_64_bytes_1[31] := PlcOutputs.ST40_1_DM260_User_Data_64_bytes_1[31];
	HwOutputs.ST40_1_DM260_User_Data_64_bytes_1[32] := PlcOutputs.ST40_1_DM260_User_Data_64_bytes_1[32];
	HwOutputs.ST40_1_DM260_User_Data_64_bytes_1[33] := PlcOutputs.ST40_1_DM260_User_Data_64_bytes_1[33];
	HwOutputs.ST40_1_DM260_User_Data_64_bytes_1[34] := PlcOutputs.ST40_1_DM260_User_Data_64_bytes_1[34];
	HwOutputs.ST40_1_DM260_User_Data_64_bytes_1[35] := PlcOutputs.ST40_1_DM260_User_Data_64_bytes_1[35];
	HwOutputs.ST40_1_DM260_User_Data_64_bytes_1[36] := PlcOutputs.ST40_1_DM260_User_Data_64_bytes_1[36];
	HwOutputs.ST40_1_DM260_User_Data_64_bytes_1[37] := PlcOutputs.ST40_1_DM260_User_Data_64_bytes_1[37];
	HwOutputs.ST40_1_DM260_User_Data_64_bytes_1[38] := PlcOutputs.ST40_1_DM260_User_Data_64_bytes_1[38];
	HwOutputs.ST40_1_DM260_User_Data_64_bytes_1[39] := PlcOutputs.ST40_1_DM260_User_Data_64_bytes_1[39];
	HwOutputs.ST40_1_DM260_User_Data_64_bytes_1[40] := PlcOutputs.ST40_1_DM260_User_Data_64_bytes_1[40];
	HwOutputs.ST40_1_DM260_User_Data_64_bytes_1[41] := PlcOutputs.ST40_1_DM260_User_Data_64_bytes_1[41];
	HwOutputs.ST40_1_DM260_User_Data_64_bytes_1[42] := PlcOutputs.ST40_1_DM260_User_Data_64_bytes_1[42];
	HwOutputs.ST40_1_DM260_User_Data_64_bytes_1[43] := PlcOutputs.ST40_1_DM260_User_Data_64_bytes_1[43];
	HwOutputs.ST40_1_DM260_User_Data_64_bytes_1[44] := PlcOutputs.ST40_1_DM260_User_Data_64_bytes_1[44];
	HwOutputs.ST40_1_DM260_User_Data_64_bytes_1[45] := PlcOutputs.ST40_1_DM260_User_Data_64_bytes_1[45];
	HwOutputs.ST40_1_DM260_User_Data_64_bytes_1[46] := PlcOutputs.ST40_1_DM260_User_Data_64_bytes_1[46];
	HwOutputs.ST40_1_DM260_User_Data_64_bytes_1[47] := PlcOutputs.ST40_1_DM260_User_Data_64_bytes_1[47];
	HwOutputs.ST40_1_DM260_User_Data_64_bytes_1[48] := PlcOutputs.ST40_1_DM260_User_Data_64_bytes_1[48];
	HwOutputs.ST40_1_DM260_User_Data_64_bytes_1[49] := PlcOutputs.ST40_1_DM260_User_Data_64_bytes_1[49];
	HwOutputs.ST40_1_DM260_User_Data_64_bytes_1[50] := PlcOutputs.ST40_1_DM260_User_Data_64_bytes_1[50];
	HwOutputs.ST40_1_DM260_User_Data_64_bytes_1[51] := PlcOutputs.ST40_1_DM260_User_Data_64_bytes_1[51];
	HwOutputs.ST40_1_DM260_User_Data_64_bytes_1[52] := PlcOutputs.ST40_1_DM260_User_Data_64_bytes_1[52];
	HwOutputs.ST40_1_DM260_User_Data_64_bytes_1[53] := PlcOutputs.ST40_1_DM260_User_Data_64_bytes_1[53];
	HwOutputs.ST40_1_DM260_User_Data_64_bytes_1[54] := PlcOutputs.ST40_1_DM260_User_Data_64_bytes_1[54];
	HwOutputs.ST40_1_DM260_User_Data_64_bytes_1[55] := PlcOutputs.ST40_1_DM260_User_Data_64_bytes_1[55];
	HwOutputs.ST40_1_DM260_User_Data_64_bytes_1[56] := PlcOutputs.ST40_1_DM260_User_Data_64_bytes_1[56];
	HwOutputs.ST40_1_DM260_User_Data_64_bytes_1[57] := PlcOutputs.ST40_1_DM260_User_Data_64_bytes_1[57];
	HwOutputs.ST40_1_DM260_User_Data_64_bytes_1[58] := PlcOutputs.ST40_1_DM260_User_Data_64_bytes_1[58];
	HwOutputs.ST40_1_DM260_User_Data_64_bytes_1[59] := PlcOutputs.ST40_1_DM260_User_Data_64_bytes_1[59];
	HwOutputs.ST40_1_DM260_User_Data_64_bytes_1[60] := PlcOutputs.ST40_1_DM260_User_Data_64_bytes_1[60];
	HwOutputs.ST40_1_DM260_User_Data_64_bytes_1[61] := PlcOutputs.ST40_1_DM260_User_Data_64_bytes_1[61];
	HwOutputs.ST40_1_DM260_User_Data_64_bytes_1[62] := PlcOutputs.ST40_1_DM260_User_Data_64_bytes_1[62];
	HwOutputs.ST40_1_DM260_User_Data_64_bytes_1[63] := PlcOutputs.ST40_1_DM260_User_Data_64_bytes_1[63];
	HwOutputs.ST40_1_DM260_User_Data_64_bytes_1[64] := PlcOutputs.ST40_1_DM260_User_Data_64_bytes_1[64];
	HwOutputs.ST40_1_DM260_User_Data_64_bytes_1[65] := PlcOutputs.ST40_1_DM260_User_Data_64_bytes_1[65];
	HwOutputs.ST40_1_DM260_User_Data_64_bytes_1[66] := PlcOutputs.ST40_1_DM260_User_Data_64_bytes_1[66];
	HwOutputs.ST40_1_DM260_User_Data_64_bytes_1[67] := PlcOutputs.ST40_1_DM260_User_Data_64_bytes_1[67];
	HwOutputs.ST40_2_Promess_Menu_30_33_Out_1 := PlcOutputs.ST40_2_Promess_Menu_30_33_Out_1;
	HwOutputs.ST40_2_Promess_Menu_30_34_Out_1 := PlcOutputs.ST40_2_Promess_Menu_30_34_Out_1;
	HwOutputs.ST40_2_Promess_Menu_30_35_Out_1 := PlcOutputs.ST40_2_Promess_Menu_30_35_Out_1;
	HwOutputs.ST40_2_Promess_Menu_30_36_Out_1 := PlcOutputs.ST40_2_Promess_Menu_30_36_Out_1;
	HwOutputs.ST40_2_Promess_Menu_30_37_Out_1 := PlcOutputs.ST40_2_Promess_Menu_30_37_Out_1;
	HwOutputs.ST40_2_Promess_Menu_30_38_Out_1 := PlcOutputs.ST40_2_Promess_Menu_30_38_Out_1;
	HwOutputs.ST40_2_Promess_Menu_30_39_Out_1 := PlcOutputs.ST40_2_Promess_Menu_30_39_Out_1;
	HwOutputs.ST40_2_Promess_Menu_30_40_Out_1 := PlcOutputs.ST40_2_Promess_Menu_30_40_Out_1;
	HwOutputs.ST40_2_Promess_Menu_30_41_Out_1 := PlcOutputs.ST40_2_Promess_Menu_30_41_Out_1;
	HwOutputs.ST40_2_Promess_Menu_30_42_Out_1 := PlcOutputs.ST40_2_Promess_Menu_30_42_Out_1;
	HwOutputs.ST40_2_Promess_Menu_30_43_Out_1 := PlcOutputs.ST40_2_Promess_Menu_30_43_Out_1;
	HwOutputs.ST40_2_Promess_Menu_30_44_Out_1 := PlcOutputs.ST40_2_Promess_Menu_30_44_Out_1;
	HwOutputs.ST40_2_Promess_Menu_30_45_Out_1 := PlcOutputs.ST40_2_Promess_Menu_30_45_Out_1;
	HwOutputs.ST40_2_Promess_Menu_30_46_Out_1 := PlcOutputs.ST40_2_Promess_Menu_30_46_Out_1;
	HwOutputs.ST40_2_Promess_Menu_30_47_Out_1 := PlcOutputs.ST40_2_Promess_Menu_30_47_Out_1;
	HwOutputs.ST40_2_Promess_Menu_30_48_Out_1 := PlcOutputs.ST40_2_Promess_Menu_30_48_Out_1;
	HwOutputs.ST40_2_Promess_Menu_30_49_Out_1 := PlcOutputs.ST40_2_Promess_Menu_30_49_Out_1;
	HwOutputs.ST40_2_Promess_Menu_30_50_Out_1 := PlcOutputs.ST40_2_Promess_Menu_30_50_Out_1;
	HwOutputs.ST40_2_Promess_Menu_30_51_Out_1 := PlcOutputs.ST40_2_Promess_Menu_30_51_Out_1;
	HwOutputs.ST40_2_Promess_Menu_30_52_Out_1 := PlcOutputs.ST40_2_Promess_Menu_30_52_Out_1;
	HwOutputs.ST40_2_Promess_Menu_30_53_Out_1 := PlcOutputs.ST40_2_Promess_Menu_30_53_Out_1;
	HwOutputs.ST40_2_Promess_Menu_30_54_Out_1 := PlcOutputs.ST40_2_Promess_Menu_30_54_Out_1;
	HwOutputs.ST40_2_Promess_Menu_30_55_Out_1 := PlcOutputs.ST40_2_Promess_Menu_30_55_Out_1;
	HwOutputs.ST40_2_Promess_Menu_30_56_Out_1 := PlcOutputs.ST40_2_Promess_Menu_30_56_Out_1;
	HwOutputs.ST40_2_Promess_Menu_30_57_Out_1 := PlcOutputs.ST40_2_Promess_Menu_30_57_Out_1;
	HwOutputs.ST40_2_Promess_Menu_30_58_Out_1 := PlcOutputs.ST40_2_Promess_Menu_30_58_Out_1;
	HwOutputs.ST40_2_Promess_Menu_30_59_Out_1 := PlcOutputs.ST40_2_Promess_Menu_30_59_Out_1;
	HwOutputs.ST40_2_Promess_Menu_30_60_Out_1 := PlcOutputs.ST40_2_Promess_Menu_30_60_Out_1;
	HwOutputs.ST40_2_Promess_Menu_30_61_Out_1 := PlcOutputs.ST40_2_Promess_Menu_30_61_Out_1;
	HwOutputs.ST40_2_Promess_Menu_30_62_Out_1 := PlcOutputs.ST40_2_Promess_Menu_30_62_Out_1;
	HwOutputs.ST40_2_Promess_Menu_30_63_Out_1 := PlcOutputs.ST40_2_Promess_Menu_30_63_Out_1;
	HwOutputs.ST40_2_Promess_Menu_30_64_Out_1 := PlcOutputs.ST40_2_Promess_Menu_30_64_Out_1;
	HwOutputs.ST40_CPX_MPA1S_VMPA1_FB_EMS_8_8DO_1 := PlcOutputs.ST40_CPX_MPA1S_VMPA1_FB_EMS_8_8DO_1;
	HwOutputs.ST40_CPX_MPA1S_VMPA1_FB_EMS_8_8DO_2 := PlcOutputs.ST40_CPX_MPA1S_VMPA1_FB_EMS_8_8DO_2;
	HwOutputs.ST40_CPX_MPA1S_VMPA1_FB_EMS_8_8DO_3 := PlcOutputs.ST40_CPX_MPA1S_VMPA1_FB_EMS_8_8DO_3;
	HwOutputs.ST40_CPX_MPA1G_VMPA1_FB_EMG_8_8DO_1 := PlcOutputs.ST40_CPX_MPA1G_VMPA1_FB_EMG_8_8DO_1;
	HwOutputs.ST40_ET200SP_CM_4xIO_Link_1[0] := PlcOutputs.ST40_ET200SP_CM_4xIO_Link_1[0];
	HwOutputs.ST40_ET200SP_CM_4xIO_Link_1[1] := PlcOutputs.ST40_ET200SP_CM_4xIO_Link_1[1];
	HwOutputs.ST40_ET200SP_CM_4xIO_Link_1[2] := PlcOutputs.ST40_ET200SP_CM_4xIO_Link_1[2];
	HwOutputs.ST40_ET200SP_CM_4xIO_Link_1[3] := PlcOutputs.ST40_ET200SP_CM_4xIO_Link_1[3];
	HwOutputs.ST40_ET200SP_CM_4xIO_Link_1[4] := PlcOutputs.ST40_ET200SP_CM_4xIO_Link_1[4];
	HwOutputs.ST40_ET200SP_CM_4xIO_Link_1[5] := PlcOutputs.ST40_ET200SP_CM_4xIO_Link_1[5];
	HwOutputs.ST40_ET200SP_CM_4xIO_Link_1[6] := PlcOutputs.ST40_ET200SP_CM_4xIO_Link_1[6];
	HwOutputs.ST40_ET200SP_CM_4xIO_Link_1[7] := PlcOutputs.ST40_ET200SP_CM_4xIO_Link_1[7];
	HwOutputs.ST40_ET200SP_CM_4xIO_Link_1[8] := PlcOutputs.ST40_ET200SP_CM_4xIO_Link_1[8];
	HwOutputs.ST40_ET200SP_CM_4xIO_Link_1[9] := PlcOutputs.ST40_ET200SP_CM_4xIO_Link_1[9];
	HwOutputs.ST40_ET200SP_CM_4xIO_Link_1[10] := PlcOutputs.ST40_ET200SP_CM_4xIO_Link_1[10];
	HwOutputs.ST40_ET200SP_CM_4xIO_Link_1[11] := PlcOutputs.ST40_ET200SP_CM_4xIO_Link_1[11];
	HwOutputs.ST40_ET200SP_CM_4xIO_Link_1[12] := PlcOutputs.ST40_ET200SP_CM_4xIO_Link_1[12];
	HwOutputs.ST40_ET200SP_CM_4xIO_Link_1[13] := PlcOutputs.ST40_ET200SP_CM_4xIO_Link_1[13];
	HwOutputs.ST40_ET200SP_CM_4xIO_Link_1[14] := PlcOutputs.ST40_ET200SP_CM_4xIO_Link_1[14];
	HwOutputs.ST40_ET200SP_CM_4xIO_Link_1[15] := PlcOutputs.ST40_ET200SP_CM_4xIO_Link_1[15];
	HwOutputs.ST40_ET200SP_CM_4xIO_Link_1[16] := PlcOutputs.ST40_ET200SP_CM_4xIO_Link_1[16];
	HwOutputs.ST40_ET200SP_CM_4xIO_Link_1[17] := PlcOutputs.ST40_ET200SP_CM_4xIO_Link_1[17];
	HwOutputs.ST40_ET200SP_CM_4xIO_Link_1[18] := PlcOutputs.ST40_ET200SP_CM_4xIO_Link_1[18];
	HwOutputs.ST40_ET200SP_CM_4xIO_Link_1[19] := PlcOutputs.ST40_ET200SP_CM_4xIO_Link_1[19];
	HwOutputs.ST40_ET200SP_CM_4xIO_Link_1[20] := PlcOutputs.ST40_ET200SP_CM_4xIO_Link_1[20];
	HwOutputs.ST40_ET200SP_CM_4xIO_Link_1[21] := PlcOutputs.ST40_ET200SP_CM_4xIO_Link_1[21];
	HwOutputs.ST40_ET200SP_CM_4xIO_Link_1[22] := PlcOutputs.ST40_ET200SP_CM_4xIO_Link_1[22];
	HwOutputs.ST40_ET200SP_CM_4xIO_Link_1[23] := PlcOutputs.ST40_ET200SP_CM_4xIO_Link_1[23];
	HwOutputs.ST40_ET200SP_CM_4xIO_Link_1[24] := PlcOutputs.ST40_ET200SP_CM_4xIO_Link_1[24];
	HwOutputs.ST40_ET200SP_CM_4xIO_Link_1[25] := PlcOutputs.ST40_ET200SP_CM_4xIO_Link_1[25];
	HwOutputs.ST40_ET200SP_CM_4xIO_Link_1[26] := PlcOutputs.ST40_ET200SP_CM_4xIO_Link_1[26];
	HwOutputs.ST40_ET200SP_CM_4xIO_Link_1[27] := PlcOutputs.ST40_ET200SP_CM_4xIO_Link_1[27];
	HwOutputs.ST40_ET200SP_CM_4xIO_Link_1[28] := PlcOutputs.ST40_ET200SP_CM_4xIO_Link_1[28];
	HwOutputs.ST40_ET200SP_CM_4xIO_Link_1[29] := PlcOutputs.ST40_ET200SP_CM_4xIO_Link_1[29];
	HwOutputs.ST40_ET200SP_CM_4xIO_Link_1[30] := PlcOutputs.ST40_ET200SP_CM_4xIO_Link_1[30];
	HwOutputs.ST40_ET200SP_CM_4xIO_Link_1[31] := PlcOutputs.ST40_ET200SP_CM_4xIO_Link_1[31];
	HwOutputs.ST40_ET200SP_CM_4xIO_Link_2[0] := PlcOutputs.ST40_ET200SP_CM_4xIO_Link_2[0];
	HwOutputs.ST40_ET200SP_CM_4xIO_Link_2[1] := PlcOutputs.ST40_ET200SP_CM_4xIO_Link_2[1];
	HwOutputs.ST40_ET200SP_CM_4xIO_Link_2[2] := PlcOutputs.ST40_ET200SP_CM_4xIO_Link_2[2];
	HwOutputs.ST40_ET200SP_CM_4xIO_Link_2[3] := PlcOutputs.ST40_ET200SP_CM_4xIO_Link_2[3];
	HwOutputs.ST40_ET200SP_CM_4xIO_Link_2[4] := PlcOutputs.ST40_ET200SP_CM_4xIO_Link_2[4];
	HwOutputs.ST40_ET200SP_CM_4xIO_Link_2[5] := PlcOutputs.ST40_ET200SP_CM_4xIO_Link_2[5];
	HwOutputs.ST40_ET200SP_CM_4xIO_Link_2[6] := PlcOutputs.ST40_ET200SP_CM_4xIO_Link_2[6];
	HwOutputs.ST40_ET200SP_CM_4xIO_Link_2[7] := PlcOutputs.ST40_ET200SP_CM_4xIO_Link_2[7];
	HwOutputs.ST40_ET200SP_CM_4xIO_Link_2[8] := PlcOutputs.ST40_ET200SP_CM_4xIO_Link_2[8];
	HwOutputs.ST40_ET200SP_CM_4xIO_Link_2[9] := PlcOutputs.ST40_ET200SP_CM_4xIO_Link_2[9];
	HwOutputs.ST40_ET200SP_CM_4xIO_Link_2[10] := PlcOutputs.ST40_ET200SP_CM_4xIO_Link_2[10];
	HwOutputs.ST40_ET200SP_CM_4xIO_Link_2[11] := PlcOutputs.ST40_ET200SP_CM_4xIO_Link_2[11];
	HwOutputs.ST40_ET200SP_CM_4xIO_Link_2[12] := PlcOutputs.ST40_ET200SP_CM_4xIO_Link_2[12];
	HwOutputs.ST40_ET200SP_CM_4xIO_Link_2[13] := PlcOutputs.ST40_ET200SP_CM_4xIO_Link_2[13];
	HwOutputs.ST40_ET200SP_CM_4xIO_Link_2[14] := PlcOutputs.ST40_ET200SP_CM_4xIO_Link_2[14];
	HwOutputs.ST40_ET200SP_CM_4xIO_Link_2[15] := PlcOutputs.ST40_ET200SP_CM_4xIO_Link_2[15];
	HwOutputs.ST40_ET200SP_CM_4xIO_Link_2[16] := PlcOutputs.ST40_ET200SP_CM_4xIO_Link_2[16];
	HwOutputs.ST40_ET200SP_CM_4xIO_Link_2[17] := PlcOutputs.ST40_ET200SP_CM_4xIO_Link_2[17];
	HwOutputs.ST40_ET200SP_CM_4xIO_Link_2[18] := PlcOutputs.ST40_ET200SP_CM_4xIO_Link_2[18];
	HwOutputs.ST40_ET200SP_CM_4xIO_Link_2[19] := PlcOutputs.ST40_ET200SP_CM_4xIO_Link_2[19];
	HwOutputs.ST40_ET200SP_CM_4xIO_Link_2[20] := PlcOutputs.ST40_ET200SP_CM_4xIO_Link_2[20];
	HwOutputs.ST40_ET200SP_CM_4xIO_Link_2[21] := PlcOutputs.ST40_ET200SP_CM_4xIO_Link_2[21];
	HwOutputs.ST40_ET200SP_CM_4xIO_Link_2[22] := PlcOutputs.ST40_ET200SP_CM_4xIO_Link_2[22];
	HwOutputs.ST40_ET200SP_CM_4xIO_Link_2[23] := PlcOutputs.ST40_ET200SP_CM_4xIO_Link_2[23];
	HwOutputs.ST40_ET200SP_CM_4xIO_Link_2[24] := PlcOutputs.ST40_ET200SP_CM_4xIO_Link_2[24];
	HwOutputs.ST40_ET200SP_CM_4xIO_Link_2[25] := PlcOutputs.ST40_ET200SP_CM_4xIO_Link_2[25];
	HwOutputs.ST40_ET200SP_CM_4xIO_Link_2[26] := PlcOutputs.ST40_ET200SP_CM_4xIO_Link_2[26];
	HwOutputs.ST40_ET200SP_CM_4xIO_Link_2[27] := PlcOutputs.ST40_ET200SP_CM_4xIO_Link_2[27];
	HwOutputs.ST40_ET200SP_CM_4xIO_Link_2[28] := PlcOutputs.ST40_ET200SP_CM_4xIO_Link_2[28];
	HwOutputs.ST40_ET200SP_CM_4xIO_Link_2[29] := PlcOutputs.ST40_ET200SP_CM_4xIO_Link_2[29];
	HwOutputs.ST40_ET200SP_CM_4xIO_Link_2[30] := PlcOutputs.ST40_ET200SP_CM_4xIO_Link_2[30];
	HwOutputs.ST40_ET200SP_CM_4xIO_Link_2[31] := PlcOutputs.ST40_ET200SP_CM_4xIO_Link_2[31];
	HwOutputs.ST40_ET200SP_DQ_16x24VDC_0_5A_ST_1 := PlcOutputs.ST40_ET200SP_DQ_16x24VDC_0_5A_ST_1;
	HwOutputs.ST40_ET200SP_DQ_8x24VDC_0_5A_ST_2 := PlcOutputs.ST40_ET200SP_DQ_8x24VDC_0_5A_ST_2;
	HwOutputs.ST40_ET200SP_DQ_8x24VDC_0_5A_ST_3 := PlcOutputs.ST40_ET200SP_DQ_8x24VDC_0_5A_ST_3;
END_FUNCTION
